C01819=1228.848,396.986,-78.994,-175.700,7.745,148.240
C01820=1228.852,396.739,-78.959,-175.700,7.743,148.239
C01821=1228.857,396.491,-78.926,-175.701,7.740,148.239
C01822=1228.860,396.243,-78.891,-175.702,7.738,148.239
C01823=1228.864,395.996,-78.857,-175.703,7.735,148.238
C01824=1228.869,395.748,-78.824,-175.703,7.733,148.238
C01825=1228.873,395.501,-78.790,-175.704,7.731,148.237
C01826=1228.876,395.253,-78.755,-175.705,7.728,148.237
C01827=1228.881,395.005,-78.722,-175.706,7.726,148.237
C01828=1228.885,394.758,-78.688,-175.707,7.723,148.236
C01829=1228.890,394.510,-78.654,-175.707,7.721,148.236
C01830=1228.893,394.262,-78.620,-175.708,7.718,148.235
C01831=1228.897,394.015,-78.586,-175.709,7.716,148.235
C01832=1228.902,393.767,-78.552,-175.710,7.713,148.234
C01833=1228.906,393.486,-78.513,-175.711,7.711,148.234
C01834=1228.911,393.204,-78.476,-175.712,7.707,148.233
C01835=1228.915,392.923,-78.437,-175.713,7.706,148.233
C01836=1228.920,392.641,-78.398,-175.714,7.703,148.233
C01837=1228.924,392.394,-78.364,-175.714,7.700,148.232
C01838=1228.928,392.147,-78.330,-175.715,7.698,148.232
C01839=1228.933,391.899,-78.297,-175.716,7.695,148.231
C01840=1228.936,391.651,-78.262,-175.717,7.692,148.231
C01841=1228.940,391.403,-78.229,-175.718,7.690,148.231
C01842=1228.945,391.156,-78.195,-175.719,7.687,148.230
C01843=1228.949,390.908,-78.161,-175.720,7.685,148.230
C01844=1228.952,390.660,-78.127,-175.721,7.682,148.229
C01845=1228.957,390.412,-78.093,-175.721,7.680,148.229
C01846=1228.961,390.165,-78.060,-175.722,7.677,148.229
C01847=1228.965,389.917,-78.026,-175.723,7.675,148.228
C01848=1228.970,389.670,-77.992,-175.724,7.672,148.228
C01849=1228.973,389.421,-77.958,-175.725,7.670,148.227
C01850=1228.977,389.174,-77.925,-175.726,7.668,148.227
C01851=1228.981,388.926,-77.891,-175.727,7.665,148.227
C01852=1228.986,388.679,-77.857,-175.728,7.663,148.226
C01853=1228.990,388.431,-77.824,-175.729,7.660,148.226
C01854=1228.993,388.183,-77.790,-175.730,7.657,148.225
C01855=1228.998,387.935,-77.756,-175.730,7.655,148.225
C01856=1229.002,387.688,-77.723,-175.731,7.652,148.225
C01857=1229.006,387.441,-77.689,-175.733,7.649,148.224
C01858=1229.010,387.193,-77.656,-175.733,7.647,148.224
C01859=1229.014,386.945,-77.621,-175.734,7.644,148.223
C01860=1229.018,386.697,-77.588,-175.736,7.642,148.223
C01861=1229.022,386.449,-77.555,-175.736,7.640,148.223
C01862=1229.026,386.202,-77.521,-175.737,7.637,148.222
C01863=1229.031,385.954,-77.487,-175.738,7.635,148.222
C01864=1229.035,385.706,-77.454,-175.739,7.632,148.222
C01865=1229.038,385.459,-77.420,-175.740,7.629,148.221
C01866=1229.042,385.211,-77.386,-175.741,7.626,148.221
C01867=1229.047,384.963,-77.353,-175.742,7.624,148.220
C01868=1229.051,384.716,-77.319,-175.743,7.622,148.220
C01869=1229.055,384.468,-77.286,-175.744,7.619,148.220
C01870=1229.059,384.220,-77.252,-175.745,7.617,148.219
C01871=1229.064,383.973,-77.218,-175.746,7.614,148.219
C01872=1229.068,383.724,-77.184,-175.747,7.611,148.218
C01873=1229.072,383.477,-77.151,-175.748,7.609,148.218
C01874=1229.075,383.230,-77.117,-175.749,7.606,148.218
C01875=1229.080,382.982,-77.084,-175.750,7.603,148.217
C01876=1229.084,382.734,-77.051,-175.752,7.601,148.217
C01877=1229.089,382.486,-77.017,-175.752,7.599,148.217
C01878=1229.092,382.239,-76.983,-175.753,7.596,148.216
C01879=1229.096,381.991,-76.950,-175.754,7.593,148.216
C01880=1229.100,381.743,-76.917,-175.756,7.590,148.215
C01881=1229.104,381.495,-76.884,-175.756,7.588,148.215
C01882=1229.108,381.248,-76.850,-175.757,7.585,148.215
C01883=1229.113,381.000,-76.816,-175.759,7.583,148.214
C01884=1229.117,380.752,-76.783,-175.760,7.580,148.214
C01885=1229.121,380.504,-76.750,-175.760,7.578,148.214
C01886=1229.125,380.257,-76.717,-175.762,7.575,148.213
C01887=1229.129,380.010,-76.683,-175.763,7.572,148.213
C01888=1229.133,379.762,-76.650,-175.764,7.570,148.213
C01889=1229.137,379.513,-76.616,-175.765,7.568,148.212
C01890=1229.142,379.265,-76.582,-175.766,7.565,148.212
C01891=1229.146,379.018,-76.549,-175.767,7.562,148.211
C01892=1229.150,378.770,-76.516,-175.768,7.559,148.211
C01893=1229.154,378.522,-76.483,-175.770,7.556,148.211
C01894=1229.158,378.275,-76.449,-175.770,7.554,148.210
C01895=1229.162,378.027,-76.416,-175.771,7.551,148.210
C01896=1229.166,377.780,-76.383,-175.773,7.549,148.210
C01897=1229.170,377.532,-76.349,-175.774,7.546,148.209
C01898=1229.175,377.284,-76.316,-175.775,7.543,148.209
C01899=1229.179,377.036,-76.283,-175.777,7.540,148.208
C01900=1229.183,376.789,-76.250,-175.777,7.539,148.208
C01901=1229.187,376.541,-76.217,-175.778,7.536,148.208
C01902=1229.191,376.293,-76.184,-175.780,7.533,148.208
C01903=1229.195,376.045,-76.150,-175.781,7.530,148.207
C01904=1229.200,375.797,-76.116,-175.782,7.528,148.207
C01905=1229.204,375.549,-76.083,-175.783,7.525,148.206
C01906=1229.208,375.301,-76.050,-175.785,7.522,148.206
C01907=1229.212,375.054,-76.017,-175.786,7.519,148.206
C01908=1229.216,374.806,-75.984,-175.787,7.517,148.205
C01909=1229.220,374.558,-75.951,-175.788,7.515,148.205
C01910=1229.224,374.310,-75.917,-175.789,7.512,148.205
C01911=1229.229,374.063,-75.884,-175.791,7.509,148.204
C01912=1229.233,373.815,-75.851,-175.792,7.506,148.204
C01913=1229.237,373.567,-75.818,-175.793,7.504,148.204
C01914=1229.241,373.320,-75.785,-175.794,7.501,148.203
C01915=1229.245,373.072,-75.752,-175.796,7.498,148.203
C01916=1229.248,372.824,-75.719,-175.797,7.495,148.203
C01917=1229.253,372.577,-75.686,-175.798,7.493,148.202
C01918=1229.257,372.329,-75.653,-175.800,7.490,148.202
C01919=1229.261,372.081,-75.620,-175.801,7.488,148.202
C01920=1229.265,371.833,-75.586,-175.802,7.485,148.201
C01921=1229.269,371.586,-75.553,-175.803,7.483,148.201
C01922=1229.274,371.337,-75.521,-175.804,7.480,148.201
C01923=1229.278,371.090,-75.488,-175.806,7.477,148.200
C01924=1229.282,370.842,-75.455,-175.807,7.474,148.200
C01925=1229.286,370.594,-75.421,-175.808,7.472,148.200
C01926=1229.290,370.346,-75.388,-175.810,7.469,148.199
C01927=1229.294,370.099,-75.355,-175.811,7.466,148.199
C01928=1229.298,369.851,-75.322,-175.812,7.463,148.199
C01929=1229.303,369.603,-75.290,-175.814,7.461,148.198
C01930=1229.306,369.355,-75.257,-175.815,7.458,148.198
C01931=1229.310,369.108,-75.224,-175.816,7.455,148.198
C01932=1229.315,368.860,-75.191,-175.818,7.453,148.198
C01933=1229.319,368.612,-75.157,-175.819,7.450,148.197
C01934=1229.324,368.364,-75.125,-175.821,7.447,148.197
C01935=1229.328,368.117,-75.092,-175.822,7.445,148.197
C01936=1229.332,367.869,-75.059,-175.823,7.442,148.196
C01937=1229.336,367.589,-75.023,-175.825,7.439,148.196
C01938=1229.341,367.309,-74.985,-175.826,7.436,148.196
C01939=1229.345,367.030,-74.948,-175.828,7.433,148.195
C01940=1229.351,366.750,-74.911,-175.830,7.429,148.195
C01941=1229.354,366.503,-74.879,-175.831,7.427,148.195
C01942=1229.358,366.255,-74.846,-175.833,7.424,148.194
C01943=1229.363,366.008,-74.812,-175.834,7.421,148.194
C01944=1229.367,365.759,-74.780,-175.835,7.419,148.194
C01945=1229.371,365.511,-74.747,-175.837,7.416,148.194
C01946=1229.375,365.264,-74.714,-175.838,7.413,148.193
C01947=1229.379,365.016,-74.682,-175.840,7.411,148.193
C01948=1229.383,364.768,-74.649,-175.841,7.408,148.193
C01949=1229.388,364.520,-74.616,-175.843,7.405,148.192
C01950=1229.392,364.272,-74.583,-175.844,7.403,148.192
C01951=1229.396,364.025,-74.551,-175.845,7.400,148.192
C01952=1229.400,363.777,-74.519,-175.847,7.398,148.192
C01953=1229.404,363.529,-74.485,-175.848,7.395,148.191
C01954=1229.409,363.281,-74.453,-175.850,7.392,148.191
C01955=1229.412,363.033,-74.420,-175.851,7.388,148.191
C01956=1229.416,362.786,-74.387,-175.853,7.386,148.190
C01957=1229.421,362.537,-74.355,-175.855,7.383,148.190
C01958=1229.424,362.290,-74.322,-175.856,7.381,148.190
C01959=1229.429,362.042,-74.290,-175.857,7.378,148.190
C01960=1229.433,361.794,-74.257,-175.859,7.375,148.189
C01961=1229.438,361.546,-74.225,-175.860,7.373,148.189
C01962=1229.441,361.299,-74.192,-175.862,7.370,148.189
C01963=1229.446,361.050,-74.160,-175.863,7.367,148.188
C01964=1229.450,360.803,-74.126,-175.865,7.365,148.188
C01965=1229.453,360.555,-74.095,-175.867,7.361,148.188
C01966=1229.458,360.308,-74.062,-175.868,7.359,148.188
C01967=1229.463,360.059,-74.029,-175.870,7.356,148.187
C01968=1229.466,359.812,-73.997,-175.871,7.354,148.187
C01969=1229.470,359.563,-73.964,-175.873,7.351,148.187
C01970=1229.475,359.315,-73.932,-175.874,7.348,148.187
C01971=1229.478,359.068,-73.899,-175.876,7.346,148.186
C01972=1229.483,358.820,-73.867,-175.877,7.343,148.186
C01973=1229.487,358.573,-73.835,-175.879,7.340,148.186
C01974=1229.491,358.324,-73.802,-175.881,7.337,148.186
C01975=1229.496,358.076,-73.770,-175.882,7.334,148.185
C01976=1229.499,357.828,-73.737,-175.884,7.332,148.185
C01977=1229.504,357.581,-73.705,-175.886,7.329,148.185
C01978=1229.507,357.333,-73.673,-175.887,7.327,148.185
C01979=1229.512,357.085,-73.640,-175.888,7.324,148.185
C01980=1229.516,356.837,-73.608,-175.890,7.321,148.184
C01981=1229.520,356.590,-73.576,-175.892,7.318,148.184
C01982=1229.525,356.342,-73.543,-175.894,7.316,148.184
C01983=1229.529,356.094,-73.511,-175.895,7.313,148.184
C01984=1229.533,355.845,-73.479,-175.896,7.310,148.183
C01985=1229.536,355.598,-73.446,-175.898,7.308,148.183
C01986=1229.541,355.350,-73.414,-175.900,7.304,148.183
C01987=1229.546,355.102,-73.382,-175.902,7.302,148.183
C01988=1229.550,354.854,-73.350,-175.904,7.299,148.183
C01989=1229.554,354.606,-73.317,-175.905,7.297,148.182
C01990=1229.558,354.359,-73.285,-175.907,7.294,148.182
C01991=1229.562,354.110,-73.253,-175.908,7.291,148.182
C01992=1229.566,353.862,-73.221,-175.910,7.288,148.182
C01993=1229.570,353.615,-73.188,-175.912,7.285,148.181
C01994=1229.575,353.367,-73.156,-175.913,7.283,148.181
C01995=1229.579,353.119,-73.124,-175.915,7.280,148.181
C01996=1229.583,352.871,-73.092,-175.917,7.278,148.181
C01997=1229.588,352.623,-73.060,-175.919,7.275,148.181
C01998=1229.592,352.375,-73.028,-175.920,7.272,148.180
C01999=1229.596,352.127,-72.995,-175.922,7.269,148.180
C02000=1229.599,351.879,-72.963,-175.924,7.267,148.180
C02001=1229.604,351.632,-72.932,-175.925,7.264,148.180
C02002=1229.608,351.384,-72.899,-175.927,7.262,148.180
C02003=1229.612,351.136,-72.867,-175.929,7.258,148.179
C02004=1229.617,350.888,-72.835,-175.931,7.256,148.179
C02005=1229.621,350.640,-72.803,-175.932,7.253,148.179
C02006=1229.625,350.392,-72.771,-175.934,7.251,148.179
C02007=1229.629,350.144,-72.739,-175.936,7.248,148.179
C02008=1229.633,349.896,-72.708,-175.938,7.245,148.178
C02009=1229.637,349.648,-72.675,-175.939,7.242,148.178
C02010=1229.642,349.401,-72.644,-175.941,7.240,148.178
C02011=1229.646,349.152,-72.611,-175.943,7.237,148.178
C02012=1229.650,348.904,-72.579,-175.945,7.234,148.178
C02013=1229.654,348.657,-72.548,-175.946,7.232,148.177
C02014=1229.659,348.409,-72.516,-175.948,7.229,148.177
C02015=1229.662,348.160,-72.484,-175.950,7.226,148.177
C02016=1229.667,347.913,-72.452,-175.951,7.224,148.177
C02017=1229.671,347.665,-72.420,-175.953,7.221,148.177
C02018=1229.675,347.417,-72.388,-175.955,7.218,148.177
C02019=1229.679,347.169,-72.356,-175.957,7.216,148.176
C02020=1229.684,346.921,-72.324,-175.958,7.213,148.176
C02021=1229.688,346.674,-72.293,-175.960,7.210,148.176
C02022=1229.692,346.426,-72.261,-175.963,7.207,148.176
C02023=1229.696,346.177,-72.228,-175.964,7.205,148.176
C02024=1229.700,345.930,-72.197,-175.966,7.202,148.176
C02025=1229.704,345.681,-72.166,-175.968,7.200,148.175
C02026=1229.709,345.433,-72.133,-175.970,7.196,148.175
C02027=1229.713,345.186,-72.102,-175.971,7.194,148.175
C02028=1229.717,344.938,-72.070,-175.973,7.191,148.175
C02029=1229.722,344.690,-72.038,-175.975,7.189,148.175
C02030=1229.726,344.442,-72.006,-175.977,7.186,148.175
C02031=1229.730,344.193,-71.975,-175.979,7.183,148.174
C02032=1229.734,343.946,-71.943,-175.980,7.181,148.174
C02033=1229.738,343.698,-71.911,-175.982,7.178,148.174
C02034=1229.743,343.450,-71.879,-175.984,7.175,148.174
C02035=1229.746,343.202,-71.848,-175.986,7.173,148.174
C02036=1229.751,342.954,-71.817,-175.988,7.170,148.174
C02037=1229.755,342.706,-71.785,-175.990,7.168,148.174
C02038=1229.760,342.459,-71.753,-175.992,7.164,148.173
C02039=1229.763,342.211,-71.721,-175.994,7.162,148.173
C02040=1229.767,341.962,-71.690,-175.995,7.159,148.173
C02041=1229.772,341.685,-71.655,-175.998,7.156,148.173
C02042=1229.777,341.408,-71.619,-175.999,7.153,148.173
C02043=1229.782,341.129,-71.584,-176.002,7.150,148.173
C02044=1229.787,340.852,-71.548,-176.004,7.147,148.172
C02045=1229.791,340.604,-71.517,-176.006,7.144,148.172
C02046=1229.795,340.356,-71.486,-176.007,7.142,148.172
C02047=1229.799,340.108,-71.454,-176.009,7.140,148.172
C02048=1229.804,339.860,-71.423,-176.012,7.136,148.172
C02049=1229.807,339.612,-71.391,-176.013,7.134,148.172
C02050=1229.812,339.365,-71.360,-176.015,7.132,148.172
C02051=1229.816,339.116,-71.328,-176.017,7.129,148.172
C02052=1229.821,338.869,-71.297,-176.019,7.126,148.171
C02053=1229.825,338.620,-71.265,-176.021,7.123,148.171
C02054=1229.829,338.373,-71.234,-176.023,7.121,148.171
C02055=1229.833,338.124,-71.203,-176.024,7.118,148.171
C02056=1229.837,337.877,-71.171,-176.027,7.115,148.171
C02057=1229.841,337.628,-71.140,-176.029,7.113,148.171
C02058=1229.846,337.381,-71.109,-176.030,7.110,148.171
C02059=1229.850,337.132,-71.078,-176.033,7.107,148.171
C02060=1229.854,336.885,-71.046,-176.035,7.105,148.170
C02061=1229.858,336.636,-71.015,-176.036,7.102,148.170
C02062=1229.862,336.389,-70.984,-176.038,7.100,148.170
C02063=1229.866,336.140,-70.952,-176.041,7.097,148.170
C02064=1229.871,335.893,-70.921,-176.043,7.094,148.170
C02065=1229.875,335.644,-70.890,-176.044,7.092,148.170
C02066=1229.879,335.397,-70.858,-176.046,7.089,148.170
C02067=1229.883,335.148,-70.827,-176.048,7.086,148.170
C02068=1229.887,334.901,-70.796,-176.050,7.084,148.170
C02069=1229.892,334.653,-70.765,-176.052,7.081,148.170
C02070=1229.896,334.404,-70.734,-176.054,7.078,148.169
C02071=1229.900,334.157,-70.702,-176.056,7.076,148.169
C02072=1229.904,333.908,-70.671,-176.058,7.073,148.169
C02073=1229.909,333.660,-70.640,-176.060,7.071,148.169
C02074=1229.912,333.412,-70.609,-176.062,7.068,148.169
C02075=1229.917,333.164,-70.578,-176.064,7.065,148.169
C02076=1229.922,332.916,-70.547,-176.066,7.063,148.169
C02077=1229.925,332.668,-70.515,-176.068,7.060,148.169
C02078=1229.930,332.420,-70.484,-176.070,7.057,148.169
C02079=1229.934,332.171,-70.453,-176.072,7.055,148.169
C02080=1229.938,331.924,-70.422,-176.074,7.053,148.169
C02081=1229.943,331.676,-70.391,-176.076,7.049,148.168
C02082=1229.947,331.427,-70.360,-176.078,7.047,148.168
C02083=1229.952,331.179,-70.329,-176.080,7.044,148.168
C02084=1229.955,330.932,-70.298,-176.082,7.042,148.168
C02085=1229.959,330.684,-70.267,-176.084,7.039,148.168
C02086=1229.964,330.436,-70.236,-176.086,7.037,148.168
C02087=1229.968,330.188,-70.206,-176.088,7.034,148.168
C02088=1229.972,329.939,-70.175,-176.091,7.031,148.168
C02089=1229.977,329.692,-70.143,-176.093,7.029,148.168
C02090=1229.981,329.443,-70.112,-176.094,7.026,148.168
C02091=1229.985,329.196,-70.082,-176.096,7.024,148.168
C02092=1229.989,328.948,-70.051,-176.099,7.021,148.168
C02093=1229.993,328.699,-70.020,-176.101,7.018,148.168
C02094=1229.998,328.451,-69.989,-176.103,7.016,148.168
C02095=1230.002,328.203,-69.958,-176.105,7.013,148.167
C02096=1230.005,327.955,-69.927,-176.107,7.011,148.167
C02097=1230.010,327.707,-69.896,-176.109,7.008,148.167
C02098=1230.015,327.459,-69.866,-176.111,7.006,148.167
C02099=1230.019,327.211,-69.835,-176.113,7.003,148.167
C02100=1230.023,326.963,-69.804,-176.115,7.000,148.167
C02101=1230.027,326.715,-69.773,-176.117,6.998,148.167
C02102=1230.032,326.467,-69.743,-176.119,6.995,148.167
C02103=1230.036,326.219,-69.712,-176.121,6.992,148.167
C02104=1230.040,325.971,-69.681,-176.124,6.990,148.167
C02105=1230.044,325.723,-69.651,-176.125,6.988,148.167
C02106=1230.048,325.474,-69.620,-176.128,6.985,148.167
C02107=1230.053,325.226,-69.589,-176.130,6.982,148.167
C02108=1230.057,324.979,-69.559,-176.132,6.980,148.167
C02109=1230.061,324.731,-69.528,-176.134,6.977,148.167
C02110=1230.065,324.482,-69.497,-176.136,6.975,148.167
C02111=1230.070,324.234,-69.466,-176.138,6.972,148.167
C02112=1230.074,323.986,-69.436,-176.141,6.969,148.167
C02113=1230.079,323.738,-69.405,-176.143,6.967,148.167
C02114=1230.083,323.490,-69.374,-176.144,6.964,148.166
C02115=1230.087,323.242,-69.344,-176.146,6.962,148.167
C02116=1230.091,322.994,-69.314,-176.149,6.959,148.166
C02117=1230.095,322.746,-69.283,-176.151,6.957,148.167
C02118=1230.099,322.497,-69.252,-176.153,6.954,148.166
C02119=1230.104,322.249,-69.222,-176.155,6.951,148.166
C02120=1230.108,322.002,-69.191,-176.157,6.949,148.166
C02121=1230.112,321.754,-69.161,-176.159,6.946,148.166
C02122=1230.117,321.505,-69.131,-176.161,6.944,148.166
C02123=1230.120,321.257,-69.100,-176.164,6.941,148.166
C02124=1230.125,321.009,-69.069,-176.166,6.939,148.166
C02125=1230.129,320.761,-69.039,-176.168,6.936,148.166
C02126=1230.134,320.513,-69.008,-176.170,6.933,148.166
C02127=1230.139,320.265,-68.978,-176.172,6.931,148.166
C02128=1230.142,320.016,-68.948,-176.174,6.929,148.166
C02129=1230.146,319.768,-68.917,-176.177,6.927,148.166
C02130=1230.150,319.521,-68.887,-176.179,6.923,148.166
C02131=1230.155,319.272,-68.857,-176.181,6.921,148.166
C02132=1230.159,319.024,-68.827,-176.183,6.919,148.166
C02133=1230.163,318.776,-68.796,-176.186,6.916,148.166
C02134=1230.167,318.528,-68.766,-176.188,6.913,148.166
C02135=1230.172,318.280,-68.735,-176.189,6.911,148.166
C02136=1230.176,318.032,-68.705,-176.191,6.909,148.166
C02137=1230.181,317.783,-68.675,-176.194,6.906,148.166
C02138=1230.185,317.536,-68.645,-176.196,6.903,148.166
C02139=1230.189,317.288,-68.614,-176.198,6.901,148.166
C02140=1230.193,317.039,-68.584,-176.201,6.898,148.166
C02141=1230.197,316.791,-68.554,-176.202,6.896,148.166
C02142=1230.202,316.543,-68.524,-176.205,6.893,148.166
C02143=1230.206,316.295,-68.493,-176.207,6.891,148.166
C02144=1230.210,316.047,-68.463,-176.209,6.888,148.166
C02145=1230.215,315.771,-68.430,-176.211,6.886,148.166
C02146=1230.220,315.496,-68.396,-176.214,6.883,148.166
C02147=1230.225,315.219,-68.363,-176.217,6.880,148.166
C02148=1230.229,314.944,-68.329,-176.219,6.878,148.166
C02149=1230.234,314.695,-68.299,-176.221,6.874,148.166
C02150=1230.238,314.448,-68.269,-176.224,6.872,148.166
C02151=1230.242,314.199,-68.239,-176.226,6.870,148.166
C02152=1230.247,313.951,-68.209,-176.227,6.867,148.166
C02153=1230.251,313.703,-68.179,-176.230,6.864,148.166
C02154=1230.256,313.455,-68.149,-176.232,6.862,148.166
C02155=1230.259,313.207,-68.119,-176.234,6.860,148.166
C02156=1230.264,312.959,-68.089,-176.237,6.857,148.166
C02157=1230.268,312.711,-68.059,-176.239,6.855,148.166
C02158=1230.272,312.462,-68.029,-176.241,6.852,148.166
C02159=1230.276,312.214,-67.999,-176.243,6.850,148.166
C02160=1230.281,311.966,-67.969,-176.246,6.847,148.166
C02161=1230.285,311.717,-67.939,-176.248,6.845,148.166
C02162=1230.289,311.470,-67.909,-176.250,6.843,148.166
C02163=1230.294,311.221,-67.879,-176.253,6.840,148.166
C02164=1230.298,310.973,-67.850,-176.255,6.837,148.166
C02165=1230.302,310.725,-67.819,-176.257,6.835,148.167
C02166=1230.307,310.477,-67.789,-176.259,6.833,148.167
C02167=1230.311,310.228,-67.760,-176.262,6.830,148.167
C02168=1230.315,309.981,-67.730,-176.264,6.828,148.167
C02169=1230.320,309.732,-67.700,-176.266,6.825,148.167
C02170=1230.324,309.484,-67.670,-176.268,6.822,148.167
C02171=1230.328,309.236,-67.641,-176.271,6.820,148.167
C02172=1230.332,308.988,-67.611,-176.273,6.818,148.167
C02173=1230.337,308.739,-67.581,-176.275,6.816,148.167
C02174=1230.341,308.491,-67.551,-176.277,6.813,148.167
C02175=1230.345,308.243,-67.522,-176.279,6.810,148.167
C02176=1230.349,307.995,-67.491,-176.282,6.808,148.167
C02177=1230.353,307.747,-67.462,-176.284,6.806,148.167
C02178=1230.358,307.498,-67.432,-176.286,6.803,148.167
C02179=1230.362,307.250,-67.403,-176.288,6.801,148.167
C02180=1230.366,307.002,-67.373,-176.291,6.799,148.167
C02181=1230.371,306.753,-67.344,-176.293,6.796,148.167
C02182=1230.375,306.507,-67.314,-176.295,6.793,148.167
C02183=1230.380,306.258,-67.284,-176.297,6.791,148.167
C02184=1230.384,306.010,-67.254,-176.300,6.789,148.167
C02185=1230.388,305.761,-67.225,-176.302,6.786,148.167
C02186=1230.393,305.513,-67.195,-176.304,6.784,148.167
C02187=1230.397,305.265,-67.166,-176.306,6.781,148.167
C02188=1230.401,305.017,-67.137,-176.308,6.779,148.167
C02189=1230.406,304.768,-67.106,-176.311,6.776,148.167
C02190=1230.410,304.520,-67.077,-176.313,6.774,148.167
C02191=1230.414,304.271,-67.048,-176.315,6.772,148.168
C02192=1230.418,304.023,-67.018,-176.318,6.770,148.168
C02193=1230.423,303.775,-66.989,-176.321,6.767,148.168
C02194=1230.427,303.527,-66.960,-176.323,6.764,148.168
C02195=1230.431,303.279,-66.930,-176.325,6.762,148.168
C02196=1230.436,303.031,-66.901,-176.327,6.760,148.168
C02197=1230.440,302.783,-66.871,-176.330,6.757,148.168
C02198=1230.444,302.534,-66.842,-176.332,6.755,148.168
C02199=1230.448,302.286,-66.812,-176.334,6.752,148.168
C02200=1230.452,302.038,-66.783,-176.336,6.750,148.168
C02201=1230.457,301.789,-66.753,-176.339,6.747,148.168
C02202=1230.462,301.541,-66.723,-176.341,6.745,148.168
C02203=1230.466,301.293,-66.694,-176.343,6.743,148.168
C02204=1230.470,301.045,-66.665,-176.345,6.741,148.169
C02205=1230.475,300.797,-66.635,-176.348,6.738,148.169
C02206=1230.479,300.548,-66.607,-176.350,6.736,148.169
C02207=1230.483,300.300,-66.577,-176.352,6.733,148.169
C02208=1230.488,300.051,-66.548,-176.355,6.731,148.169
C02209=1230.492,299.804,-66.519,-176.357,6.728,148.169
C02210=1230.496,299.556,-66.489,-176.360,6.726,148.169
C02211=1230.500,299.308,-66.460,-176.362,6.724,148.169
C02212=1230.504,299.059,-66.432,-176.364,6.722,148.169
C02213=1230.509,298.810,-66.402,-176.367,6.719,148.169
C02214=1230.513,298.563,-66.373,-176.369,6.717,148.169
C02215=1230.518,298.315,-66.344,-176.371,6.714,148.169
C02216=1230.522,298.066,-66.314,-176.373,6.712,148.170
C02217=1230.526,297.817,-66.285,-176.376,6.709,148.170
C02218=1230.530,297.569,-66.256,-176.378,6.707,148.170
C02219=1230.535,297.321,-66.226,-176.381,6.705,148.170
C02220=1230.540,297.073,-66.198,-176.383,6.703,148.170
C02221=1230.544,296.824,-66.169,-176.385,6.700,148.170
C02222=1230.548,296.576,-66.139,-176.387,6.698,148.170
C02223=1230.551,296.328,-66.110,-176.390,6.696,148.170
C02224=1230.557,296.080,-66.082,-176.392,6.693,148.170
C02225=1230.561,295.832,-66.053,-176.394,6.691,148.170
C02226=1230.565,295.583,-66.024,-176.397,6.688,148.170
C02227=1230.569,295.335,-65.994,-176.399,6.686,148.171
C02228=1230.574,295.087,-65.965,-176.402,6.684,148.171
C02229=1230.579,294.838,-65.936,-176.404,6.682,148.171
C02230=1230.582,294.590,-65.908,-176.406,6.679,148.171
C02231=1230.586,294.342,-65.878,-176.409,6.677,148.171
C02232=1230.591,294.094,-65.850,-176.411,6.675,148.171
C02233=1230.596,293.846,-65.820,-176.413,6.672,148.171
C02234=1230.600,293.597,-65.792,-176.415,6.670,148.171
C02235=1230.604,293.349,-65.763,-176.418,6.667,148.171
C02236=1230.609,293.100,-65.734,-176.420,6.665,148.172
C02237=1230.613,292.852,-65.705,-176.423,6.663,148.172
C02238=1230.617,292.603,-65.676,-176.425,6.661,148.172
C02239=1230.621,292.356,-65.648,-176.428,6.658,148.172
C02240=1230.626,292.107,-65.619,-176.430,6.656,148.172
C02241=1230.630,291.859,-65.590,-176.432,6.654,148.172
C02242=1230.635,291.611,-65.561,-176.435,6.652,148.172
C02243=1230.639,291.363,-65.532,-176.437,6.649,148.172
C02244=1230.643,291.114,-65.504,-176.439,6.646,148.172
C02245=1230.647,290.866,-65.474,-176.442,6.644,148.173
C02246=1230.652,290.617,-65.446,-176.444,6.642,148.173
C02247=1230.656,290.369,-65.418,-176.446,6.640,148.173
C02248=1230.661,290.121,-65.388,-176.448,6.638,148.173
C02249=1230.666,289.847,-65.357,-176.451,6.635,148.173
C02250=1230.670,289.573,-65.325,-176.454,6.633,148.173
C02251=1230.675,289.298,-65.294,-176.457,6.630,148.173
C02252=1230.680,289.024,-65.261,-176.459,6.627,148.173
C02253=1230.684,288.777,-65.233,-176.462,6.625,148.174
C02254=1230.689,288.528,-65.205,-176.464,6.623,148.174
C02255=1230.692,288.280,-65.176,-176.466,6.621,148.174
C02256=1230.697,288.032,-65.147,-176.469,6.619,148.174
C02257=1230.702,287.783,-65.119,-176.471,6.616,148.174
C02258=1230.706,287.535,-65.091,-176.473,6.614,148.174
C02259=1230.710,287.287,-65.061,-176.476,6.612,148.174
C02260=1230.715,287.038,-65.033,-176.478,6.609,148.175
C02261=1230.719,286.790,-65.005,-176.481,6.608,148.175
C02262=1230.723,286.541,-64.976,-176.483,6.605,148.175
C02263=1230.727,286.294,-64.948,-176.486,6.602,148.175
C02264=1230.732,286.045,-64.919,-176.488,6.600,148.175
C02265=1230.736,285.796,-64.891,-176.490,6.598,148.175
C02266=1230.741,285.548,-64.862,-176.492,6.596,148.175
C02267=1230.745,285.299,-64.834,-176.495,6.594,148.176
C02268=1230.749,285.052,-64.805,-176.498,6.591,148.176
C02269=1230.754,284.803,-64.777,-176.500,6.589,148.176
C02270=1230.758,284.555,-64.749,-176.502,6.587,148.176
C02271=1230.763,284.306,-64.720,-176.504,6.585,148.176
C02272=1230.767,284.058,-64.692,-176.507,6.583,148.176
C02273=1230.771,283.809,-64.663,-176.509,6.580,148.176
C02274=1230.775,283.561,-64.635,-176.512,6.578,148.177
C02275=1230.780,283.313,-64.607,-176.514,6.576,148.177
C02276=1230.784,283.064,-64.579,-176.517,6.574,148.177
C02277=1230.789,282.817,-64.550,-176.519,6.571,148.177
C02278=1230.793,282.568,-64.522,-176.521,6.569,148.177
C02279=1230.798,282.320,-64.493,-176.524,6.567,148.177
C02280=1230.801,282.071,-64.465,-176.526,6.564,148.177
C02281=1230.807,281.823,-64.437,-176.529,6.562,148.178
C02282=1230.810,281.574,-64.409,-176.531,6.560,148.178
C02283=1230.815,281.327,-64.381,-176.534,6.558,148.178
C02284=1230.819,281.078,-64.352,-176.536,6.556,148.178
C02285=1230.823,280.830,-64.324,-176.538,6.554,148.178
C02286=1230.828,280.581,-64.296,-176.541,6.551,148.178
C02287=1230.832,280.333,-64.268,-176.543,6.549,148.178
C02288=1230.836,280.084,-64.240,-176.546,6.547,148.179
C02289=1230.841,279.836,-64.212,-176.548,6.545,148.179
C02290=1230.845,279.587,-64.184,-176.550,6.543,148.179
C02291=1230.850,279.339,-64.155,-176.553,6.541,148.179
C02292=1230.854,279.090,-64.127,-176.556,6.538,148.179
C02293=1230.858,278.842,-64.100,-176.558,6.536,148.179
C02294=1230.863,278.594,-64.071,-176.560,6.534,148.180
C02295=1230.867,278.346,-64.043,-176.563,6.532,148.180
C02296=1230.872,278.098,-64.015,-176.565,6.530,148.180
C02297=1230.876,277.848,-63.987,-176.567,6.527,148.180
C02298=1230.881,277.600,-63.959,-176.570,6.526,148.181
C02299=1230.884,277.352,-63.931,-176.573,6.522,148.181
C02300=1230.890,277.104,-63.903,-176.575,6.521,148.181
C02301=1230.893,276.855,-63.875,-176.577,6.518,148.181
C02302=1230.898,276.607,-63.847,-176.580,6.516,148.181
C02303=1230.902,276.359,-63.820,-176.582,6.514,148.181
C02304=1230.907,276.110,-63.791,-176.585,6.512,148.182
C02305=1230.911,275.862,-63.763,-176.587,6.510,148.182
C02306=1230.915,275.613,-63.735,-176.589,6.508,148.182
C02307=1230.920,275.365,-63.708,-176.592,6.505,148.182
C02308=1230.925,275.117,-63.680,-176.595,6.503,148.182
C02309=1230.928,274.868,-63.652,-176.597,6.501,148.182
C02310=1230.933,274.620,-63.625,-176.599,6.499,148.183
C02311=1230.938,274.371,-63.596,-176.601,6.497,148.183
C02312=1230.942,274.123,-63.568,-176.604,6.495,148.183
C02313=1230.947,273.874,-63.541,-176.606,6.493,148.183
C02314=1230.950,273.626,-63.513,-176.609,6.491,148.183
C02315=1230.955,273.378,-63.485,-176.611,6.488,148.183
C02316=1230.960,273.129,-63.458,-176.614,6.486,148.184
C02317=1230.964,272.881,-63.429,-176.617,6.484,148.184
C02318=1230.968,272.633,-63.402,-176.619,6.482,148.184
C02319=1230.972,272.383,-63.374,-176.621,6.480,148.184
C02320=1230.977,272.136,-63.346,-176.623,6.478,148.184
C02321=1230.981,271.887,-63.319,-176.626,6.476,148.185
C02322=1230.986,271.638,-63.291,-176.628,6.474,148.185
C02323=1230.990,271.390,-63.264,-176.631,6.472,148.185
C02324=1230.995,271.142,-63.236,-176.634,6.469,148.185
C02325=1230.999,270.893,-63.209,-176.636,6.467,148.185
C02326=1231.003,270.645,-63.181,-176.639,6.465,148.186
C02327=1231.008,270.396,-63.153,-176.641,6.463,148.186
C02328=1231.012,270.148,-63.126,-176.643,6.461,148.186
C02329=1231.016,269.899,-63.098,-176.645,6.459,148.186
C02330=1231.021,269.651,-63.070,-176.648,6.457,148.186
C02331=1231.026,269.402,-63.043,-176.651,6.455,148.187
C02332=1231.030,269.154,-63.015,-176.653,6.453,148.187
C02333=1231.034,268.905,-62.988,-176.655,6.451,148.187
C02334=1231.039,268.658,-62.960,-176.658,6.448,148.187
C02335=1231.043,268.409,-62.933,-176.661,6.446,148.187
C02336=1231.047,268.160,-62.905,-176.663,6.444,148.188
C02337=1231.052,267.912,-62.878,-176.665,6.442,148.188
C02338=1231.056,267.663,-62.851,-176.668,6.440,148.188
C02339=1231.061,267.416,-62.823,-176.670,6.438,148.188
C02340=1231.065,267.166,-62.795,-176.673,6.436,148.188
C02341=1231.069,266.918,-62.768,-176.675,6.434,148.189
C02342=1231.074,266.670,-62.740,-176.677,6.432,148.189
C02343=1231.078,266.422,-62.713,-176.680,6.430,148.189
C02344=1231.083,266.172,-62.686,-176.682,6.427,148.189
C02345=1231.087,265.924,-62.658,-176.685,6.426,148.189
C02346=1231.092,265.676,-62.631,-176.687,6.424,148.190
C02347=1231.096,265.427,-62.604,-176.690,6.421,148.190
C02348=1231.101,265.179,-62.577,-176.692,6.419,148.190
C02349=1231.105,264.930,-62.549,-176.695,6.417,148.190
C02350=1231.109,264.682,-62.522,-176.697,6.415,148.190
C02351=1231.114,264.433,-62.495,-176.700,6.413,148.191
C02352=1231.119,264.185,-62.468,-176.702,6.411,148.191
C02353=1231.123,263.913,-62.438,-176.704,6.409,148.191
C02354=1231.128,263.640,-62.408,-176.708,6.406,148.191
C02355=1231.132,263.367,-62.378,-176.710,6.404,148.192
C02356=1231.137,263.095,-62.348,-176.713,6.402,148.192
C02357=1231.141,262.846,-62.321,-176.715,6.400,148.192
C02358=1231.146,262.598,-62.294,-176.718,6.398,148.192
C02359=1231.151,262.349,-62.267,-176.720,6.396,148.193
C02360=1231.155,262.101,-62.240,-176.723,6.393,148.193
C02361=1231.160,261.852,-62.213,-176.725,6.391,148.193
C02362=1231.163,261.603,-62.186,-176.728,6.389,148.193
C02363=1231.168,261.355,-62.158,-176.730,6.387,148.193
C02364=1231.172,261.107,-62.131,-176.733,6.385,148.194
C02365=1231.177,260.858,-62.104,-176.735,6.383,148.194
C02366=1231.182,260.610,-62.077,-176.738,6.381,148.194
C02367=1231.186,260.361,-62.050,-176.740,6.379,148.194
C02368=1231.190,260.113,-62.023,-176.743,6.377,148.195
C02369=1231.194,259.864,-61.996,-176.745,6.375,148.195
C02370=1231.199,259.616,-61.969,-176.747,6.373,148.195
C02371=1231.204,259.367,-61.942,-176.750,6.371,148.195
C02372=1231.208,259.119,-61.915,-176.753,6.369,148.196
C02373=1231.212,258.870,-61.888,-176.755,6.367,148.196
C02374=1231.217,258.622,-61.861,-176.757,6.365,148.196
C02375=1231.222,258.373,-61.834,-176.760,6.363,148.196
C02376=1231.226,258.125,-61.807,-176.762,6.361,148.196
C02377=1231.230,257.877,-61.781,-176.765,6.359,148.197
C02378=1231.235,257.628,-61.753,-176.767,6.357,148.197
C02379=1231.239,257.379,-61.726,-176.770,6.355,148.197
C02380=1231.244,257.131,-61.699,-176.772,6.353,148.197
C02381=1231.248,256.882,-61.673,-176.775,6.351,148.198
C02382=1231.252,256.633,-61.646,-176.777,6.349,148.198
C02383=1231.257,256.385,-61.619,-176.779,6.347,148.198
C02384=1231.261,256.137,-61.593,-176.782,6.345,148.198
C02385=1231.266,255.888,-61.566,-176.785,6.343,148.199
C02386=1231.270,255.640,-61.539,-176.787,6.342,148.199
C02387=1231.274,255.391,-61.512,-176.789,6.339,148.199
C02388=1231.279,255.142,-61.486,-176.792,6.337,148.199
C02389=1231.284,254.894,-61.459,-176.794,6.336,148.200
C02390=1231.288,254.646,-61.432,-176.797,6.334,148.200
C02391=1231.292,254.397,-61.405,-176.799,6.332,148.200
C02392=1231.297,254.149,-61.378,-176.802,6.330,148.200
C02393=1231.301,253.900,-61.352,-176.804,6.328,148.201
C02394=1231.306,253.651,-61.325,-176.807,6.326,148.201
C02395=1231.311,253.403,-61.298,-176.809,6.324,148.201
C02396=1231.315,253.155,-61.272,-176.812,6.322,148.201
C02397=1231.319,252.905,-61.245,-176.814,6.320,148.202
C02398=1231.323,252.657,-61.219,-176.817,6.318,148.202
C02399=1231.328,252.409,-61.192,-176.819,6.316,148.202
C02400=1231.333,252.160,-61.165,-176.822,6.314,148.202
C02401=1231.337,251.912,-61.139,-176.824,6.312,148.203
C02402=1231.342,251.663,-61.112,-176.827,6.310,148.203
C02403=1231.346,251.415,-61.085,-176.829,6.308,148.203
C02404=1231.350,251.166,-61.059,-176.832,6.306,148.203
C02405=1231.354,250.918,-61.033,-176.834,6.304,148.204
C02406=1231.359,250.668,-61.006,-176.837,6.302,148.204
C02407=1231.363,250.420,-60.980,-176.839,6.300,148.204
C02408=1231.368,250.172,-60.953,-176.842,6.298,148.204
C02409=1231.372,249.923,-60.927,-176.844,6.296,148.205
C02410=1231.377,249.674,-60.900,-176.847,6.294,148.205
C02411=1231.381,249.426,-60.874,-176.849,6.292,148.205
C02412=1231.386,249.177,-60.847,-176.852,6.290,148.205
C02413=1231.390,248.929,-60.821,-176.854,6.288,148.206
C02414=1231.395,248.681,-60.795,-176.857,6.287,148.206
C02415=1231.399,248.432,-60.768,-176.859,6.285,148.206
C02416=1231.404,248.183,-60.742,-176.862,6.283,148.207
C02417=1231.408,247.935,-60.715,-176.864,6.281,148.207
C02418=1231.413,247.686,-60.689,-176.867,6.279,148.207
C02419=1231.417,247.438,-60.663,-176.869,6.277,148.207
C02420=1231.422,247.189,-60.636,-176.872,6.275,148.208
C02421=1231.426,246.940,-60.610,-176.875,6.273,148.208
C02422=1231.430,246.692,-60.584,-176.877,6.271,148.208
C02423=1231.435,246.443,-60.558,-176.879,6.269,148.208
C02424=1231.439,246.195,-60.532,-176.882,6.267,148.209
C02425=1231.444,245.946,-60.505,-176.885,6.265,148.209
C02426=1231.448,245.698,-60.479,-176.887,6.263,148.209
C02427=1231.453,245.449,-60.453,-176.890,6.261,148.210
C02428=1231.457,245.200,-60.426,-176.892,6.259,148.210
C02429=1231.461,244.952,-60.400,-176.894,6.257,148.210
C02430=1231.466,244.703,-60.375,-176.897,6.255,148.210
C02431=1231.470,244.454,-60.347,-176.900,6.254,148.211
C02432=1231.475,244.206,-60.322,-176.902,6.252,148.211
C02433=1231.479,243.957,-60.296,-176.904,6.250,148.211
C02434=1231.484,243.709,-60.269,-176.906,6.248,148.211
C02435=1231.488,243.460,-60.244,-176.909,6.246,148.212
C02436=1231.492,243.211,-60.218,-176.912,6.245,148.212
C02437=1231.497,242.963,-60.191,-176.914,6.243,148.212
C02438=1231.502,242.715,-60.165,-176.917,6.241,148.213
C02439=1231.506,242.466,-60.140,-176.920,6.239,148.213
C02440=1231.511,242.217,-60.113,-176.922,6.237,148.213
C02441=1231.515,241.969,-60.087,-176.924,6.235,148.213
C02442=1231.519,241.720,-60.061,-176.927,6.233,148.214
C02443=1231.524,241.472,-60.036,-176.930,6.231,148.214
C02444=1231.529,241.223,-60.009,-176.932,6.229,148.214
C02445=1231.533,240.974,-59.984,-176.935,6.227,148.215
C02446=1231.537,240.726,-59.957,-176.937,6.225,148.215
C02447=1231.541,240.477,-59.931,-176.939,6.223,148.215
C02448=1231.547,240.228,-59.905,-176.942,6.222,148.215
C02449=1231.551,239.980,-59.880,-176.944,6.220,148.216
C02450=1231.555,239.731,-59.854,-176.947,6.218,148.216
C02451=1231.560,239.482,-59.828,-176.949,6.217,148.216
C02452=1231.565,239.234,-59.801,-176.952,6.215,148.217
C02453=1231.569,238.985,-59.776,-176.955,6.213,148.217
C02454=1231.573,238.737,-59.750,-176.957,6.211,148.217
C02455=1231.578,238.488,-59.724,-176.959,6.209,148.217
C02456=1231.582,238.240,-59.699,-176.962,6.207,148.218
C02457=1231.587,237.968,-59.671,-176.965,6.205,148.218
C02458=1231.592,237.697,-59.642,-176.967,6.203,148.218
C02459=1231.597,237.425,-59.614,-176.970,6.201,148.219
C02460=1231.602,237.153,-59.586,-176.973,6.198,148.219
C02461=1231.607,236.905,-59.560,-176.975,6.197,148.219
C02462=1231.611,236.656,-59.534,-176.978,6.196,148.220
C02463=1231.616,236.407,-59.509,-176.980,6.194,148.220
C02464=1231.620,236.159,-59.483,-176.983,6.192,148.220
C02465=1231.625,235.910,-59.458,-176.986,6.190,148.220
C02466=1231.629,235.662,-59.432,-176.988,6.188,148.221
C02467=1231.634,235.414,-59.406,-176.991,6.186,148.221
C02468=1231.638,235.165,-59.381,-176.993,6.184,148.221
C02469=1231.642,234.916,-59.355,-176.996,6.182,148.222
C02470=1231.647,234.667,-59.329,-176.998,6.180,148.222
C02471=1231.652,234.419,-59.303,-177.001,6.178,148.222
C02472=1231.656,234.170,-59.277,-177.003,6.177,148.223
C02473=1231.660,233.921,-59.252,-177.005,6.175,148.223
C02474=1231.665,233.673,-59.226,-177.008,6.174,148.223
C02475=1231.669,233.424,-59.201,-177.011,6.172,148.223
C02476=1231.674,233.175,-59.176,-177.013,6.170,148.224
C02477=1231.679,232.927,-59.150,-177.016,6.168,148.224
C02478=1231.683,232.678,-59.124,-177.018,6.166,148.224
C02479=1231.688,232.430,-59.099,-177.021,6.164,148.225
C02480=1231.692,232.181,-59.073,-177.024,6.162,148.225
C02481=1231.696,231.932,-59.048,-177.026,6.161,148.225
C02482=1231.701,231.683,-59.023,-177.028,6.159,148.226
C02483=1231.706,231.435,-58.997,-177.031,6.157,148.226
C02484=1231.710,231.186,-58.971,-177.033,6.155,148.226
C02485=1231.715,230.938,-58.946,-177.036,6.153,148.226
C02486=1231.719,230.688,-58.921,-177.038,6.152,148.227
C02487=1231.724,230.440,-58.896,-177.041,6.150,148.227
C02488=1231.728,230.191,-58.870,-177.044,6.148,148.227
C02489=1231.732,229.943,-58.844,-177.046,6.147,148.228
C02490=1231.738,229.694,-58.819,-177.048,6.145,148.228
C02491=1231.741,229.445,-58.794,-177.051,6.143,148.228
C02492=1231.746,229.197,-58.769,-177.054,6.141,148.229
C02493=1231.750,228.948,-58.743,-177.056,6.139,148.229
C02494=1231.755,228.700,-58.718,-177.059,6.137,148.229
C02495=1231.759,228.451,-58.693,-177.061,6.135,148.230
C02496=1231.764,228.202,-58.668,-177.064,6.134,148.230
C02497=1231.769,227.953,-58.642,-177.066,6.133,148.230
C02498=1231.773,227.705,-58.617,-177.069,6.131,148.231
C02499=1231.778,227.456,-58.592,-177.071,6.129,148.231
C02500=1231.782,227.207,-58.567,-177.074,6.127,148.231
C02501=1231.786,226.959,-58.541,-177.077,6.125,148.232
C02502=1231.791,226.710,-58.516,-177.079,6.123,148.232
C02503=1231.796,226.462,-58.491,-177.082,6.121,148.232
C02504=1231.800,226.212,-58.466,-177.083,6.120,148.232
C02505=1231.805,225.964,-58.440,-177.086,6.118,148.233
C02506=1231.809,225.715,-58.416,-177.089,6.116,148.233
C02507=1231.813,225.466,-58.390,-177.091,6.114,148.233
C02508=1231.818,225.218,-58.366,-177.094,6.112,148.234
C02509=1231.823,224.969,-58.340,-177.097,6.111,148.234
C02510=1231.828,224.720,-58.315,-177.099,6.109,148.234
C02511=1231.831,224.472,-58.290,-177.101,6.108,148.235
C02512=1231.836,224.223,-58.265,-177.104,6.106,148.235
C02513=1231.841,223.974,-58.240,-177.106,6.104,148.235
C02514=1231.846,223.725,-58.215,-177.109,6.102,148.236
C02515=1231.850,223.478,-58.190,-177.112,6.100,148.236
C02516=1231.854,223.228,-58.165,-177.114,6.098,148.236
C02517=1231.859,222.980,-58.140,-177.117,6.096,148.237
C02518=1231.864,222.731,-58.115,-177.119,6.095,148.237
C02519=1231.868,222.483,-58.090,-177.122,6.094,148.237
C02520=1231.872,222.233,-58.065,-177.124,6.092,148.238
C02521=1231.877,221.985,-58.040,-177.127,6.090,148.238
C02522=1231.881,221.736,-58.015,-177.130,6.088,148.238
C02523=1231.886,221.487,-57.990,-177.132,6.086,148.239
C02524=1231.891,221.238,-57.965,-177.134,6.085,148.239
C02525=1231.895,220.990,-57.940,-177.137,6.083,148.239
C02526=1231.900,220.741,-57.916,-177.139,6.081,148.240
C02527=1231.904,220.492,-57.891,-177.142,6.079,148.240
C02528=1231.909,220.244,-57.865,-177.145,6.078,148.241
C02529=1231.913,219.995,-57.841,-177.148,6.076,148.241
C02530=1231.918,219.746,-57.816,-177.150,6.075,148.241
C02531=1231.922,219.498,-57.791,-177.153,6.073,148.242
C02532=1231.927,219.249,-57.767,-177.155,6.071,148.242
C02533=1231.932,219.000,-57.742,-177.158,6.069,148.242
C02534=1231.936,218.751,-57.717,-177.160,6.067,148.243
C02535=1231.940,218.503,-57.692,-177.163,6.066,148.243
C02536=1231.945,218.254,-57.667,-177.165,6.065,148.243
C02537=1231.949,218.005,-57.643,-177.168,6.063,148.244
C02538=1231.954,217.756,-57.618,-177.170,6.061,148.244
C02539=1231.958,217.507,-57.594,-177.173,6.059,148.244
C02540=1231.963,217.259,-57.568,-177.176,6.057,148.245
C02541=1231.967,217.011,-57.544,-177.178,6.055,148.245
C02542=1231.972,216.761,-57.519,-177.180,6.054,148.245
C02543=1231.977,216.513,-57.495,-177.183,6.052,148.246
C02544=1231.981,216.263,-57.470,-177.186,6.050,148.246
C02545=1231.986,216.015,-57.446,-177.188,6.049,148.246
C02546=1231.990,215.767,-57.421,-177.191,6.047,148.247
C02547=1231.995,215.518,-57.396,-177.193,6.045,148.247
C02548=1231.999,215.269,-57.372,-177.195,6.044,148.247
C02549=1232.004,215.020,-57.347,-177.199,6.042,148.248
C02550=1232.008,214.771,-57.323,-177.201,6.040,148.248
C02551=1232.013,214.523,-57.298,-177.204,6.039,148.249
C02552=1232.018,214.274,-57.274,-177.206,6.037,148.249
C02553=1232.022,214.025,-57.249,-177.209,6.036,148.249
C02554=1232.026,213.776,-57.225,-177.211,6.034,148.250
C02555=1232.032,213.528,-57.200,-177.214,6.032,148.250
C02556=1232.036,213.279,-57.176,-177.216,6.030,148.250
C02557=1232.041,213.030,-57.151,-177.219,6.028,148.251
C02558=1232.045,212.781,-57.127,-177.221,6.027,148.251
C02559=1232.049,212.533,-57.103,-177.224,6.025,148.251
C02560=1232.054,212.284,-57.078,-177.226,6.023,148.252
C02561=1232.059,212.013,-57.051,-177.230,6.022,148.252
C02562=1232.063,211.743,-57.025,-177.232,6.020,148.252
C02563=1232.069,211.473,-56.999,-177.235,6.018,148.253
C02564=1232.073,211.202,-56.972,-177.237,6.016,148.253
C02565=1232.078,210.953,-56.948,-177.240,6.014,148.253
C02566=1232.083,210.705,-56.923,-177.243,6.013,148.254
C02567=1232.087,210.456,-56.899,-177.245,6.012,148.254
C02568=1232.092,210.207,-56.874,-177.248,6.010,148.255
C02569=1232.096,209.958,-56.850,-177.250,6.008,148.255
C02570=1232.101,209.709,-56.827,-177.253,6.006,148.255
C02571=1232.106,209.461,-56.802,-177.256,6.004,148.256
C02572=1232.110,209.212,-56.778,-177.258,6.003,148.256
C02573=1232.114,208.963,-56.753,-177.260,6.002,148.256
C02574=1232.119,208.714,-56.729,-177.263,6.000,148.257
C02575=1232.124,208.466,-56.705,-177.266,5.998,148.257
C02576=1232.128,208.217,-56.681,-177.268,5.997,148.258
C02577=1232.133,207.968,-56.656,-177.271,5.995,148.258
C02578=1232.137,207.719,-56.632,-177.274,5.993,148.258
C02579=1232.142,207.471,-56.608,-177.276,5.992,148.259
C02580=1232.147,207.221,-56.584,-177.279,5.990,148.259
C02581=1232.152,206.973,-56.560,-177.281,5.989,148.259
C02582=1232.155,206.724,-56.536,-177.284,5.987,148.260
C02583=1232.160,206.475,-56.511,-177.286,5.985,148.260
C02584=1232.165,206.226,-56.488,-177.289,5.983,148.260
C02585=1232.170,205.978,-56.463,-177.291,5.982,148.261
C02586=1232.174,205.729,-56.439,-177.294,5.980,148.261
C02587=1232.179,205.480,-56.416,-177.297,5.979,148.262
C02588=1232.183,205.231,-56.391,-177.299,5.977,148.262
C02589=1232.188,204.982,-56.367,-177.301,5.976,148.262
C02590=1232.192,204.733,-56.344,-177.304,5.974,148.263
C02591=1232.197,204.485,-56.319,-177.307,5.972,148.263
C02592=1232.202,204.236,-56.295,-177.309,5.970,148.263
C02593=1232.207,203.987,-56.271,-177.312,5.969,148.264
C02594=1232.211,203.739,-56.247,-177.314,5.968,148.264
C02595=1232.215,203.490,-56.223,-177.317,5.966,148.265
C02596=1232.219,203.241,-56.200,-177.319,5.965,148.265
C02597=1232.224,202.992,-56.176,-177.322,5.963,148.265
C02598=1232.229,202.743,-56.152,-177.324,5.961,148.266
C02599=1232.234,202.494,-56.127,-177.327,5.959,148.266
C02600=1232.238,202.245,-56.104,-177.330,5.958,148.267
C02601=1232.243,201.997,-56.080,-177.332,5.957,148.267
C02602=1232.248,201.748,-56.057,-177.335,5.955,148.267
C02603=1232.252,201.500,-56.033,-177.337,5.953,148.268
C02604=1232.256,201.250,-56.008,-177.340,5.952,148.268
C02605=1232.261,201.001,-55.984,-177.342,5.950,148.268
C02606=1232.266,200.752,-55.961,-177.345,5.948,148.269
C02607=1232.270,200.504,-55.937,-177.347,5.947,148.269
C02608=1232.275,200.255,-55.913,-177.350,5.946,148.270
C02609=1232.279,200.006,-55.889,-177.353,5.944,148.270
C02610=1232.284,199.757,-55.866,-177.355,5.942,148.270
C02611=1232.288,199.509,-55.842,-177.357,5.941,148.271
C02612=1232.293,199.260,-55.819,-177.360,5.939,148.271
C02613=1232.298,199.011,-55.794,-177.363,5.937,148.272
C02614=1232.302,198.762,-55.771,-177.365,5.936,148.272
C02615=1232.307,198.513,-55.748,-177.368,5.935,148.272
C02616=1232.311,198.265,-55.724,-177.371,5.933,148.273
C02617=1232.316,198.016,-55.700,-177.373,5.931,148.273
C02618=1232.320,197.767,-55.676,-177.375,5.930,148.273
C02619=1232.325,197.518,-55.653,-177.378,5.928,148.274
C02620=1232.330,197.269,-55.630,-177.381,5.926,148.274
C02621=1232.334,197.020,-55.605,-177.383,5.925,148.275
C02622=1232.338,196.771,-55.582,-177.386,5.924,148.275
C02623=1232.343,196.522,-55.558,-177.388,5.922,148.275
C02624=1232.348,196.273,-55.535,-177.390,5.921,148.276
C02625=1232.352,196.025,-55.511,-177.394,5.919,148.276
C02626=1232.357,195.776,-55.488,-177.396,5.917,148.277
C02627=1232.361,195.527,-55.464,-177.398,5.916,148.277
C02628=1232.366,195.278,-55.440,-177.401,5.914,148.277
C02629=1232.371,195.029,-55.417,-177.404,5.913,148.278
C02630=1232.376,194.781,-55.394,-177.406,5.912,148.278
C02631=1232.381,194.532,-55.370,-177.409,5.910,148.279
C02632=1232.385,194.283,-55.346,-177.411,5.908,148.279
C02633=1232.390,194.034,-55.323,-177.414,5.906,148.279
C02634=1232.394,193.785,-55.300,-177.416,5.905,148.280
C02635=1232.399,193.536,-55.276,-177.419,5.903,148.280
C02636=1232.404,193.287,-55.253,-177.422,5.902,148.281
C02637=1232.408,193.038,-55.230,-177.424,5.901,148.281
C02638=1232.412,192.790,-55.206,-177.427,5.899,148.281
C02639=1232.417,192.541,-55.183,-177.429,5.897,148.282
C02640=1232.422,192.292,-55.159,-177.431,5.896,148.282
C02641=1232.426,192.043,-55.136,-177.434,5.895,148.283
C02642=1232.431,191.794,-55.113,-177.437,5.893,148.283
C02643=1232.436,191.545,-55.089,-177.439,5.892,148.283
C02644=1232.440,191.296,-55.066,-177.442,5.890,148.284
C02645=1232.445,191.047,-55.043,-177.444,5.889,148.284
C02646=1232.449,190.799,-55.019,-177.447,5.887,148.285
C02647=1232.454,190.551,-54.996,-177.450,5.886,148.285
C02648=1232.459,190.302,-54.973,-177.452,5.885,148.285
C02649=1232.463,190.052,-54.949,-177.454,5.883,148.286
C02650=1232.468,189.803,-54.926,-177.458,5.881,148.286
C02651=1232.472,189.555,-54.903,-177.460,5.880,148.287
C02652=1232.477,189.306,-54.880,-177.462,5.878,148.287
C02653=1232.481,189.057,-54.857,-177.465,5.876,148.287
C02654=1232.486,188.808,-54.833,-177.467,5.875,148.288
C02655=1232.491,188.559,-54.810,-177.470,5.874,148.288
C02656=1232.495,188.311,-54.787,-177.473,5.872,148.289
C02657=1232.500,188.062,-54.764,-177.475,5.871,148.289
C02658=1232.505,187.813,-54.741,-177.477,5.869,148.289
C02659=1232.510,187.563,-54.717,-177.481,5.868,148.290
C02660=1232.513,187.315,-54.695,-177.483,5.867,148.290
C02661=1232.518,187.065,-54.672,-177.485,5.865,148.291
C02662=1232.523,186.816,-54.649,-177.487,5.864,148.291
C02663=1232.528,186.568,-54.626,-177.491,5.862,148.292
C02664=1232.532,186.319,-54.603,-177.493,5.860,148.292
C02665=1232.538,186.049,-54.578,-177.495,5.859,148.292
C02666=1232.543,185.779,-54.553,-177.498,5.858,148.293
C02667=1232.548,185.510,-54.528,-177.501,5.856,148.293
C02668=1232.552,185.240,-54.502,-177.504,5.854,148.294
C02669=1232.558,184.991,-54.480,-177.507,5.853,148.294
C02670=1232.562,184.743,-54.457,-177.509,5.852,148.295
C02671=1232.566,184.493,-54.434,-177.512,5.850,148.295
C02672=1232.571,184.244,-54.410,-177.514,5.849,148.295
C02673=1232.575,183.996,-54.388,-177.517,5.847,148.296
C02674=1232.581,183.747,-54.365,-177.519,5.845,148.296
C02675=1232.585,183.498,-54.343,-177.522,5.844,148.297
C02676=1232.589,183.249,-54.319,-177.525,5.843,148.297
C02677=1232.594,183.000,-54.296,-177.527,5.842,148.298
C02678=1232.598,182.751,-54.273,-177.529,5.840,148.298
C02679=1232.604,182.502,-54.251,-177.532,5.838,148.298
C02680=1232.608,182.254,-54.228,-177.535,5.837,148.299
C02681=1232.612,182.005,-54.205,-177.537,5.836,148.299
C02682=1232.617,181.755,-54.182,-177.539,5.835,148.300
C02683=1232.622,181.507,-54.160,-177.542,5.833,148.300
C02684=1232.626,181.258,-54.136,-177.545,5.831,148.301
C02685=1232.631,181.009,-54.114,-177.547,5.830,148.301
C02686=1232.635,180.759,-54.091,-177.550,5.828,148.301
C02687=1232.640,180.511,-54.069,-177.552,5.827,148.302
C02688=1232.645,180.262,-54.046,-177.555,5.826,148.302
C02689=1232.650,180.013,-54.023,-177.558,5.824,148.303
C02690=1232.654,179.764,-54.000,-177.560,5.823,148.303
C02691=1232.659,179.515,-53.978,-177.563,5.822,148.304
C02692=1232.663,179.266,-53.955,-177.565,5.820,148.304
C02693=1232.668,179.017,-53.931,-177.568,5.819,148.304
C02694=1232.673,178.769,-53.910,-177.570,5.817,148.305
C02695=1232.678,178.520,-53.886,-177.573,5.816,148.305
C02696=1232.682,178.270,-53.864,-177.576,5.814,148.306
C02697=1232.687,178.022,-53.841,-177.578,5.813,148.306
C02698=1232.691,177.773,-53.819,-177.581,5.812,148.307
C02699=1232.696,177.524,-53.796,-177.583,5.811,148.307
C02700=1232.700,177.274,-53.774,-177.586,5.809,148.307
C02701=1232.705,177.026,-53.751,-177.588,5.807,148.308
C02702=1232.710,176.777,-53.728,-177.591,5.806,148.308
C02703=1232.714,176.528,-53.706,-177.593,5.805,148.309
C02704=1232.719,176.279,-53.684,-177.596,5.804,148.309
C02705=1232.723,176.030,-53.661,-177.599,5.802,148.310
C02706=1232.728,175.781,-53.638,-177.601,5.801,148.310
C02707=1232.733,175.533,-53.616,-177.603,5.799,148.310
C02708=1232.737,175.283,-53.594,-177.606,5.798,148.311
C02709=1232.742,175.034,-53.571,-177.609,5.797,148.311
C02710=1232.747,174.786,-53.549,-177.611,5.795,148.312
C02711=1232.752,174.537,-53.526,-177.613,5.794,148.312
C02712=1232.756,174.288,-53.504,-177.616,5.792,148.313
C02713=1232.761,174.039,-53.482,-177.619,5.791,148.313
C02714=1232.765,173.790,-53.458,-177.621,5.789,148.313
C02715=1232.770,173.541,-53.437,-177.624,5.789,148.314
C02716=1232.775,173.292,-53.413,-177.626,5.787,148.314
C02717=1232.779,173.042,-53.391,-177.629,5.786,148.315
C02718=1232.784,172.794,-53.370,-177.632,5.784,148.315
C02719=1232.789,172.545,-53.346,-177.634,5.783,148.316
C02720=1232.794,172.296,-53.325,-177.636,5.782,148.316
C02721=1232.798,172.047,-53.303,-177.639,5.781,148.317
C02722=1232.803,171.799,-53.280,-177.642,5.779,148.317
C02723=1232.807,171.549,-53.258,-177.644,5.777,148.317
C02724=1232.812,171.300,-53.235,-177.647,5.777,148.318
C02725=1232.817,171.051,-53.214,-177.650,5.775,148.318
C02726=1232.821,170.802,-53.190,-177.652,5.774,148.319
C02727=1232.826,170.554,-53.169,-177.655,5.772,148.319
C02728=1232.830,170.304,-53.147,-177.657,5.771,148.320
C02729=1232.836,170.055,-53.124,-177.660,5.769,148.320
C02730=1232.840,169.807,-53.102,-177.662,5.769,148.321
C02731=1232.844,169.557,-53.080,-177.665,5.767,148.321
C02732=1232.849,169.309,-53.058,-177.667,5.766,148.322
C02733=1232.854,169.059,-53.035,-177.670,5.764,148.322
C02734=1232.859,168.811,-53.013,-177.672,5.763,148.322
C02735=1232.863,168.562,-52.991,-177.675,5.761,148.323
C02736=1232.868,168.313,-52.969,-177.677,5.761,148.323
C02737=1232.873,168.063,-52.947,-177.680,5.759,148.324
C02738=1232.878,167.815,-52.925,-177.682,5.758,148.324
C02739=1232.882,167.565,-52.903,-177.685,5.756,148.325
C02740=1232.887,167.317,-52.881,-177.687,5.755,148.325
C02741=1232.891,167.068,-52.858,-177.690,5.754,148.326
C02742=1232.896,166.819,-52.837,-177.693,5.753,148.326
C02743=1232.901,166.570,-52.814,-177.695,5.751,148.327
C02744=1232.906,166.321,-52.792,-177.697,5.750,148.327
C02745=1232.910,166.072,-52.770,-177.700,5.749,148.328
C02746=1232.915,165.823,-52.749,-177.703,5.748,148.328
C02747=1232.919,165.574,-52.727,-177.706,5.746,148.328
C02748=1232.924,165.325,-52.705,-177.708,5.745,148.329
C02749=1232.929,165.075,-52.682,-177.710,5.743,148.329
C02750=1232.934,164.827,-52.661,-177.713,5.743,148.330
C02751=1232.938,164.577,-52.639,-177.716,5.741,148.330
C02752=1232.943,164.329,-52.617,-177.718,5.740,148.331
C02753=1232.947,164.079,-52.595,-177.721,5.738,148.331
C02754=1232.952,163.831,-52.573,-177.723,5.737,148.332
C02755=1232.956,163.581,-52.551,-177.726,5.735,148.332
C02756=1232.961,163.333,-52.529,-177.728,5.735,148.333
C02757=1232.965,163.083,-52.507,-177.731,5.733,148.333
C02758=1232.970,162.835,-52.486,-177.734,5.732,148.334
C02759=1232.976,162.586,-52.463,-177.736,5.730,148.334
C02760=1232.980,162.336,-52.441,-177.738,5.729,148.334
C02761=1232.985,162.088,-52.420,-177.741,5.728,148.335
C02762=1232.989,161.838,-52.398,-177.744,5.727,148.335
C02763=1232.994,161.590,-52.376,-177.747,5.725,148.336
C02764=1232.998,161.341,-52.354,-177.749,5.724,148.336
C02765=1233.003,161.092,-52.332,-177.751,5.723,148.337
C02766=1233.008,160.843,-52.310,-177.754,5.722,148.337
C02767=1233.013,160.593,-52.289,-177.756,5.721,148.338
C02768=1233.018,160.345,-52.267,-177.759,5.719,148.338
C02769=1233.023,160.076,-52.243,-177.762,5.718,148.339
C02770=1233.028,159.807,-52.221,-177.765,5.717,148.339
C02771=1233.033,159.537,-52.197,-177.767,5.715,148.340
C02772=1233.037,159.268,-52.173,-177.770,5.714,148.340
C02773=1233.042,159.020,-52.152,-177.772,5.713,148.341
C02774=1233.047,158.770,-52.131,-177.775,5.712,148.341
C02775=1233.051,158.521,-52.109,-177.778,5.710,148.342
C02776=1233.056,158.272,-52.087,-177.780,5.709,148.342
C02777=1233.061,158.024,-52.065,-177.783,5.708,148.343
C02778=1233.065,157.774,-52.044,-177.785,5.707,148.343
C02779=1233.070,157.525,-52.022,-177.788,5.705,148.344
C02780=1233.075,157.277,-52.001,-177.790,5.704,148.344
C02781=1233.079,157.027,-51.979,-177.793,5.702,148.344
C02782=1233.085,156.778,-51.958,-177.795,5.702,148.345
C02783=1233.090,156.529,-51.936,-177.798,5.701,148.345
C02784=1233.094,156.280,-51.914,-177.801,5.699,148.346
C02785=1233.099,156.031,-51.892,-177.803,5.698,148.346
C02786=1233.104,155.782,-51.871,-177.806,5.697,148.347
C02787=1233.107,155.533,-51.850,-177.808,5.696,148.347
C02788=1233.112,155.284,-51.828,-177.811,5.694,148.348
C02789=1233.117,155.035,-51.807,-177.813,5.693,148.348
C02790=1233.122,154.786,-51.785,-177.815,5.692,148.349
C02791=1233.127,154.537,-51.764,-177.819,5.691,148.349
C02792=1233.132,154.288,-51.742,-177.821,5.690,148.350
C02793=1233.136,154.039,-51.720,-177.824,5.688,148.350
C02794=1233.140,153.790,-51.700,-177.826,5.687,148.351
C02795=1233.145,153.541,-51.678,-177.829,5.685,148.351
C02796=1233.150,153.292,-51.657,-177.831,5.685,148.352
C02797=1233.155,153.042,-51.635,-177.833,5.684,148.352
C02798=1233.160,152.794,-51.614,-177.836,5.682,148.353
C02799=1233.165,152.544,-51.593,-177.839,5.681,148.353
C02800=1233.168,152.295,-51.571,-177.842,5.680,148.354
C02801=1233.173,152.046,-51.550,-177.844,5.679,148.354
C02802=1233.178,151.798,-51.529,-177.846,5.678,148.354
C02803=1233.184,151.548,-51.508,-177.849,5.676,148.355
C02804=1233.188,151.299,-51.486,-177.851,5.675,148.355
C02805=1233.192,151.050,-51.465,-177.854,5.674,148.356
C02806=1233.197,150.801,-51.444,-177.856,5.673,148.356
C02807=1233.202,150.552,-51.423,-177.859,5.672,148.357
C02808=1233.207,150.303,-51.401,-177.862,5.670,148.357
C02809=1233.211,150.054,-51.380,-177.864,5.670,148.358
C02810=1233.216,149.805,-51.358,-177.867,5.668,148.358
C02811=1233.221,149.556,-51.337,-177.870,5.667,148.359
C02812=1233.225,149.308,-51.316,-177.872,5.666,148.359
C02813=1233.230,149.058,-51.295,-177.874,5.664,148.360
C02814=1233.235,148.808,-51.274,-177.877,5.664,148.360
C02815=1233.240,148.560,-51.252,-177.880,5.662,148.361
C02816=1233.244,148.311,-51.232,-177.882,5.661,148.361
C02817=1233.249,148.062,-51.210,-177.884,5.660,148.362
C02818=1233.254,147.812,-51.189,-177.887,5.659,148.362
C02819=1233.258,147.563,-51.169,-177.890,5.658,148.363
C02820=1233.263,147.315,-51.147,-177.893,5.656,148.363
C02821=1233.268,147.065,-51.126,-177.895,5.655,148.364
C02822=1233.273,146.816,-51.106,-177.897,5.655,148.364
C02823=1233.277,146.568,-51.084,-177.900,5.653,148.365
C02824=1233.282,146.318,-51.063,-177.903,5.652,148.365
C02825=1233.286,146.069,-51.042,-177.905,5.651,148.366
C02826=1233.291,145.820,-51.021,-177.908,5.650,148.366
C02827=1233.296,145.571,-51.000,-177.910,5.649,148.367
C02828=1233.301,145.322,-50.979,-177.913,5.647,148.367
C02829=1233.306,145.073,-50.958,-177.915,5.646,148.368
C02830=1233.310,144.824,-50.937,-177.917,5.645,148.368
C02831=1233.315,144.574,-50.916,-177.921,5.644,148.369
C02832=1233.319,144.325,-50.895,-177.923,5.643,148.369
C02833=1233.324,144.077,-50.874,-177.925,5.642,148.370
C02834=1233.329,143.828,-50.853,-177.928,5.640,148.370
C02835=1233.334,143.579,-50.832,-177.930,5.639,148.371
C02836=1233.339,143.329,-50.811,-177.933,5.638,148.371
C02837=1233.343,143.080,-50.791,-177.936,5.637,148.372
C02838=1233.348,142.831,-50.769,-177.938,5.636,148.372
C02839=1233.352,142.582,-50.749,-177.941,5.635,148.373
C02840=1233.357,142.333,-50.728,-177.943,5.634,148.373
C02841=1233.362,142.084,-50.707,-177.946,5.633,148.374
C02842=1233.367,141.835,-50.686,-177.948,5.631,148.374
C02843=1233.372,141.585,-50.665,-177.951,5.630,148.375
C02844=1233.376,141.337,-50.644,-177.953,5.629,148.375
C02845=1233.381,141.088,-50.623,-177.956,5.628,148.376
C02846=1233.386,140.839,-50.603,-177.958,5.627,148.376
C02847=1233.391,140.590,-50.582,-177.961,5.626,148.377
C02848=1233.395,140.340,-50.561,-177.964,5.624,148.377
C02849=1233.400,140.091,-50.540,-177.966,5.624,148.378
C02850=1233.404,139.842,-50.520,-177.968,5.623,148.378
C02851=1233.409,139.593,-50.500,-177.971,5.621,148.379
C02852=1233.414,139.344,-50.479,-177.974,5.620,148.379
C02853=1233.418,139.095,-50.458,-177.976,5.620,148.380
C02854=1233.424,138.845,-50.437,-177.979,5.618,148.380
C02855=1233.428,138.596,-50.417,-177.981,5.617,148.381
C02856=1233.433,138.347,-50.396,-177.984,5.616,148.381
C02857=1233.438,138.098,-50.376,-177.987,5.615,148.382
C02858=1233.443,137.849,-50.355,-177.989,5.614,148.382
C02859=1233.447,137.600,-50.334,-177.991,5.613,148.383
C02860=1233.452,137.351,-50.314,-177.995,5.612,148.384
C02861=1233.457,137.102,-50.293,-177.997,5.611,148.384
C02862=1233.461,136.853,-50.273,-177.999,5.610,148.385
C02863=1233.466,136.604,-50.252,-178.002,5.608,148.385
C02864=1233.471,136.355,-50.231,-178.005,5.608,148.386
C02865=1233.475,136.106,-50.211,-178.007,5.607,148.386
C02866=1233.481,135.856,-50.190,-178.010,5.605,148.387
C02867=1233.485,135.607,-50.169,-178.012,5.604,148.387
C02868=1233.489,135.359,-50.149,-178.015,5.603,148.388
C02869=1233.495,135.109,-50.128,-178.017,5.602,148.388
C02870=1233.499,134.860,-50.108,-178.020,5.601,148.389
C02871=1233.505,134.610,-50.088,-178.022,5.600,148.389
C02872=1233.509,134.361,-50.067,-178.025,5.599,148.390
C02873=1233.514,134.093,-50.045,-178.028,5.598,148.390
C02874=1233.518,133.824,-50.023,-178.030,5.597,148.391
C02875=1233.524,133.555,-50.001,-178.033,5.595,148.391
C02876=1233.529,133.287,-49.978,-178.036,5.595,148.392
C02877=1233.534,133.038,-49.958,-178.038,5.593,148.392
C02878=1233.538,132.789,-49.938,-178.041,5.592,148.393
C02879=1233.544,132.539,-49.918,-178.043,5.592,148.394
C02880=1233.548,132.290,-49.897,-178.046,5.590,148.394
C02881=1233.553,132.041,-49.877,-178.049,5.589,148.395
C02882=1233.558,131.792,-49.857,-178.051,5.588,148.395
C02883=1233.562,131.543,-49.836,-178.054,5.587,148.396
C02884=1233.567,131.294,-49.816,-178.056,5.586,148.396
C02885=1233.572,131.045,-49.796,-178.059,5.585,148.397
C02886=1233.577,130.796,-49.776,-178.061,5.584,148.397
C02887=1233.582,130.547,-49.755,-178.064,5.583,148.398
C02888=1233.586,130.298,-49.735,-178.067,5.582,148.398
C02889=1233.591,130.049,-49.714,-178.069,5.581,148.399
C02890=1233.595,129.799,-49.695,-178.072,5.580,148.399
C02891=1233.601,129.550,-49.674,-178.074,5.579,148.400
C02892=1233.605,129.301,-49.653,-178.077,5.578,148.400
C02893=1233.610,129.051,-49.634,-178.079,5.577,148.401
C02894=1233.614,128.802,-49.613,-178.082,5.576,148.402
C02895=1233.619,128.554,-49.593,-178.084,5.575,148.402
C02896=1233.625,128.304,-49.573,-178.087,5.574,148.403
C02897=1233.629,128.055,-49.553,-178.089,5.573,148.403
C02898=1233.634,127.806,-49.532,-178.092,5.571,148.404
C02899=1233.638,127.557,-49.513,-178.094,5.571,148.404
C02900=1233.643,127.308,-49.492,-178.097,5.570,148.405
C02901=1233.648,127.058,-49.473,-178.100,5.568,148.405
C02902=1233.653,126.809,-49.452,-178.102,5.568,148.406
C02903=1233.658,126.561,-49.432,-178.104,5.567,148.406
C02904=1233.663,126.311,-49.412,-178.107,5.566,148.407
C02905=1233.667,126.062,-49.392,-178.110,5.564,148.407
C02906=1233.672,125.813,-49.372,-178.112,5.564,148.408
C02907=1233.676,125.564,-49.352,-178.114,5.563,148.408
C02908=1233.681,125.314,-49.332,-178.117,5.562,148.409
C02909=1233.686,125.066,-49.312,-178.120,5.561,148.410
C02910=1233.691,124.816,-49.292,-178.122,5.560,148.410
C02911=1233.696,124.567,-49.271,-178.125,5.559,148.411
C02912=1233.701,124.317,-49.252,-178.127,5.558,148.411
C02913=1233.705,124.069,-49.231,-178.130,5.557,148.412
C02914=1233.710,123.820,-49.212,-178.133,5.556,148.412
C02915=1233.715,123.571,-49.192,-178.135,5.555,148.413
C02916=1233.720,123.321,-49.172,-178.138,5.554,148.413
C02917=1233.724,123.072,-49.152,-178.140,5.552,148.414
C02918=1233.729,122.823,-49.132,-178.143,5.552,148.414
C02919=1233.734,122.574,-49.112,-178.145,5.551,148.415
C02920=1233.739,122.325,-49.092,-178.148,5.550,148.415
C02921=1233.743,122.075,-49.073,-178.151,5.549,148.416
C02922=1233.748,121.826,-49.052,-178.153,5.548,148.416
C02923=1233.752,121.577,-49.033,-178.155,5.547,148.417
C02924=1233.757,121.329,-49.013,-178.158,5.546,148.418
C02925=1233.762,121.079,-48.993,-178.160,5.546,148.418
C02926=1233.767,120.829,-48.973,-178.163,5.544,148.419
C02927=1233.771,120.580,-48.953,-178.165,5.543,148.419
C02928=1233.777,120.332,-48.934,-178.168,5.542,148.420
C02929=1233.781,120.082,-48.914,-178.171,5.542,148.420
C02930=1233.786,119.833,-48.894,-178.173,5.540,148.421
C02931=1233.791,119.583,-48.874,-178.176,5.539,148.421
C02932=1233.796,119.335,-48.855,-178.179,5.539,148.422
C02933=1233.800,119.086,-48.834,-178.181,5.538,148.423
C02934=1233.805,118.836,-48.815,-178.184,5.536,148.423
C02935=1233.811,118.587,-48.795,-178.186,5.535,148.424
C02936=1233.815,118.338,-48.775,-178.189,5.535,148.424
C02937=1233.820,118.089,-48.755,-178.191,5.534,148.425
C02938=1233.824,117.839,-48.736,-178.193,5.533,148.425
C02939=1233.829,117.591,-48.717,-178.196,5.532,148.426
C02940=1233.833,117.342,-48.697,-178.199,5.531,148.426
C02941=1233.838,117.092,-48.677,-178.201,5.530,148.427
C02942=1233.844,116.843,-48.658,-178.204,5.529,148.428
C02943=1233.848,116.594,-48.638,-178.206,5.528,148.428
C02944=1233.853,116.344,-48.618,-178.209,5.527,148.429
C02945=1233.858,116.096,-48.598,-178.212,5.526,148.429
C02946=1233.863,115.846,-48.579,-178.214,5.525,148.430
C02947=1233.867,115.597,-48.560,-178.216,5.525,148.430
C02948=1233.872,115.348,-48.540,-178.219,5.524,148.431
C02949=1233.877,115.099,-48.521,-178.222,5.522,148.431
C02950=1233.882,114.849,-48.501,-178.224,5.522,148.432
C02951=1233.887,114.601,-48.481,-178.227,5.521,148.433
C02952=1233.891,114.351,-48.461,-178.229,5.520,148.433
C02953=1233.896,114.102,-48.442,-178.232,5.519,148.434
C02954=1233.901,113.853,-48.423,-178.234,5.518,148.434
C02955=1233.906,113.603,-48.403,-178.237,5.517,148.435
C02956=1233.910,113.354,-48.384,-178.240,5.516,148.435
C02957=1233.916,113.105,-48.364,-178.242,5.515,148.436
C02958=1233.920,112.855,-48.345,-178.244,5.515,148.436
C02959=1233.924,112.606,-48.326,-178.248,5.513,148.437
C02960=1233.930,112.357,-48.306,-178.250,5.512,148.437
C02961=1233.934,112.108,-48.286,-178.252,5.512,148.438
C02962=1233.940,111.860,-48.267,-178.255,5.511,148.439
C02963=1233.944,111.610,-48.248,-178.257,5.510,148.439
C02964=1233.948,111.361,-48.228,-178.260,5.509,148.440
C02965=1233.954,111.112,-48.209,-178.263,5.508,148.440
C02966=1233.958,110.862,-48.189,-178.265,5.507,148.441
C02967=1233.963,110.614,-48.170,-178.267,5.506,148.441
C02968=1233.968,110.364,-48.151,-178.270,5.506,148.442
C02969=1233.972,110.115,-48.131,-178.272,5.505,148.443
C02970=1233.978,109.866,-48.112,-178.275,5.503,148.443
C02971=1233.982,109.616,-48.093,-178.278,5.503,148.444
C02972=1233.987,109.367,-48.074,-178.280,5.502,148.444
C02973=1233.992,109.117,-48.054,-178.283,5.501,148.445
C02974=1233.997,108.869,-48.036,-178.285,5.501,148.445
C02975=1234.002,108.619,-48.016,-178.287,5.500,148.446
C02976=1234.006,108.370,-47.996,-178.291,5.498,148.447
C02977=1234.012,108.102,-47.976,-178.293,5.497,148.447
C02978=1234.017,107.833,-47.955,-178.296,5.497,148.448
C02979=1234.021,107.565,-47.935,-178.299,5.495,148.448
C02980=1234.027,107.296,-47.914,-178.302,5.495,148.449
C02981=1234.032,107.047,-47.895,-178.304,5.494,148.449
C02982=1234.037,106.798,-47.875,-178.306,5.493,148.450
C02983=1234.041,106.549,-47.857,-178.309,5.493,148.451
C02984=1234.046,106.300,-47.837,-178.311,5.492,148.451
C02985=1234.051,106.050,-47.817,-178.314,5.490,148.452
C02986=1234.056,105.801,-47.799,-178.317,5.490,148.452
C02987=1234.061,105.551,-47.780,-178.319,5.489,148.453
C02988=1234.065,105.303,-47.761,-178.322,5.488,148.454
C02989=1234.070,105.053,-47.741,-178.324,5.487,148.454
C02990=1234.075,104.804,-47.722,-178.326,5.486,148.455
C02991=1234.080,104.554,-47.704,-178.329,5.486,148.455
C02992=1234.085,104.306,-47.684,-178.332,5.484,148.456
C02993=1234.089,104.056,-47.665,-178.335,5.484,148.457
C02994=1234.094,103.807,-47.646,-178.337,5.483,148.457
C02995=1234.099,103.558,-47.628,-178.340,5.482,148.458
C02996=1234.104,103.309,-47.608,-178.342,5.481,148.458
C02997=1234.109,103.060,-47.589,-178.344,5.480,148.459
C02998=1234.113,102.811,-47.570,-178.347,5.480,148.459
C02999=1234.119,102.561,-47.551,-178.350,5.478,148.460
C03000=1234.123,102.312,-47.532,-178.352,5.477,148.460
C03001=1234.128,102.063,-47.513,-178.355,5.477,148.461
C03002=1234.133,101.813,-47.495,-178.357,5.476,148.462
C03003=1234.138,101.564,-47.475,-178.360,5.476,148.462
C03004=1234.142,101.315,-47.456,-178.362,5.475,148.463
C03005=1234.148,101.065,-47.438,-178.365,5.474,148.463
C03006=1234.152,100.816,-47.419,-178.367,5.473,148.464
C03007=1234.157,100.567,-47.399,-178.370,5.472,148.464
C03008=1234.162,100.318,-47.381,-178.373,5.471,148.465
C03009=1234.167,100.069,-47.362,-178.375,5.470,148.466
C03010=1234.171,99.819,-47.344,-178.378,5.470,148.466
C03011=1234.176,99.570,-47.324,-178.380,5.469,148.467
C03012=1234.181,99.321,-47.305,-178.383,5.468,148.467
C03013=1234.186,99.071,-47.287,-178.385,5.468,148.468
C03014=1234.190,98.823,-47.268,-178.387,5.467,148.468
C03015=1234.195,98.573,-47.250,-178.391,5.465,148.469
C03016=1234.200,98.324,-47.230,-178.393,5.464,148.470
C03017=1234.205,98.075,-47.212,-178.396,5.464,148.470
C03018=1234.210,97.825,-47.193,-178.398,5.463,148.471
C03019=1234.214,97.577,-47.174,-178.401,5.462,148.471
C03020=1234.220,97.327,-47.155,-178.403,5.462,148.472
C03021=1234.224,97.078,-47.136,-178.405,5.461,148.473
C03022=1234.229,96.829,-47.118,-178.408,5.460,148.473
C03023=1234.234,96.580,-47.099,-178.411,5.459,148.474
C03024=1234.239,96.330,-47.081,-178.413,5.459,148.474
C03025=1234.244,96.081,-47.061,-178.416,5.457,148.475
C03026=1234.248,95.831,-47.043,-178.419,5.456,148.476
C03027=1234.253,95.582,-47.025,-178.421,5.456,148.476
C03028=1234.259,95.333,-47.006,-178.424,5.455,148.477
C03029=1234.263,95.083,-46.987,-178.426,5.454,148.477
C03030=1234.267,94.835,-46.969,-178.428,5.454,148.478
C03031=1234.273,94.585,-46.950,-178.431,5.453,148.479
C03032=1234.277,94.336,-46.931,-178.434,5.452,148.479
C03033=1234.282,94.087,-46.913,-178.436,5.451,148.480
C03034=1234.288,93.837,-46.894,-178.438,5.451,148.480
C03035=1234.292,93.588,-46.875,-178.441,5.450,148.481
C03036=1234.297,93.339,-46.857,-178.444,5.449,148.482
C03037=1234.302,93.090,-46.838,-178.446,5.448,148.482
C03038=1234.306,92.840,-46.820,-178.449,5.447,148.483
C03039=1234.311,92.591,-46.802,-178.452,5.447,148.483
C03040=1234.316,92.342,-46.783,-178.454,5.446,148.484
C03041=1234.321,92.092,-46.764,-178.456,5.445,148.484
C03042=1234.326,91.843,-46.746,-178.459,5.444,148.485
C03043=1234.330,91.594,-46.727,-178.462,5.444,148.486
C03044=1234.336,91.345,-46.709,-178.464,5.443,148.486
C03045=1234.340,91.095,-46.691,-178.466,5.442,148.487
C03046=1234.345,90.846,-46.672,-178.469,5.442,148.487
C03047=1234.350,90.597,-46.654,-178.472,5.441,148.488
C03048=1234.355,90.347,-46.635,-178.474,5.440,148.489
C03049=1234.360,90.098,-46.617,-178.477,5.439,148.489
C03050=1234.364,89.849,-46.598,-178.480,5.438,148.490
C03051=1234.369,89.600,-46.580,-178.482,5.437,148.490
C03052=1234.374,89.350,-46.562,-178.485,5.437,148.491
C03053=1234.379,89.101,-46.543,-178.487,5.436,148.491
C03054=1234.384,88.852,-46.525,-178.490,5.435,148.492
C03055=1234.389,88.603,-46.507,-178.492,5.435,148.493
C03056=1234.393,88.353,-46.488,-178.495,5.434,148.493
C03057=1234.398,88.104,-46.470,-178.497,5.433,148.494
C03058=1234.404,87.855,-46.452,-178.500,5.432,148.495
C03059=1234.408,87.606,-46.433,-178.502,5.432,148.495
C03060=1234.413,87.356,-46.415,-178.505,5.431,148.496
C03061=1234.417,87.107,-46.397,-178.507,5.431,148.497
C03062=1234.422,86.858,-46.379,-178.510,5.430,148.497
C03063=1234.427,86.609,-46.361,-178.512,5.429,148.498
C03064=1234.432,86.358,-46.342,-178.515,5.428,148.498
C03065=1234.437,86.110,-46.323,-178.517,5.428,148.499
C03066=1234.442,85.861,-46.305,-178.521,5.426,148.500
C03067=1234.447,85.612,-46.287,-178.523,5.425,148.500
C03068=1234.452,85.362,-46.269,-178.525,5.425,148.501
C03069=1234.456,85.112,-46.251,-178.528,5.424,148.501
C03070=1234.461,84.863,-46.233,-178.531,5.424,148.502
C03071=1234.466,84.614,-46.215,-178.533,5.423,148.502
C03072=1234.471,84.365,-46.196,-178.535,5.422,148.503
C03073=1234.476,84.115,-46.178,-178.538,5.421,148.504
C03074=1234.481,83.866,-46.160,-178.541,5.421,148.504
C03075=1234.486,83.616,-46.142,-178.543,5.420,148.505
C03076=1234.490,83.367,-46.124,-178.545,5.419,148.505
C03077=1234.495,83.118,-46.106,-178.548,5.419,148.506
C03078=1234.500,82.869,-46.088,-178.551,5.418,148.507
C03079=1234.505,82.620,-46.070,-178.553,5.418,148.507
C03080=1234.510,82.371,-46.052,-178.556,5.417,148.508
C03081=1234.515,82.102,-46.032,-178.558,5.416,148.509
C03082=1234.520,81.833,-46.013,-178.561,5.416,148.509
C03083=1234.526,81.565,-45.993,-178.564,5.414,148.510
C03084=1234.531,81.297,-45.974,-178.567,5.414,148.511
C03085=1234.536,81.047,-45.956,-178.569,5.413,148.511
C03086=1234.540,80.798,-45.938,-178.572,5.412,148.512
C03087=1234.545,80.549,-45.920,-178.574,5.412,148.512
C03088=1234.550,80.300,-45.902,-178.577,5.411,148.513
C03089=1234.555,80.051,-45.884,-178.580,5.410,148.514
C03090=1234.560,79.801,-45.866,-178.582,5.409,148.514
C03091=1234.565,79.552,-45.848,-178.584,5.409,148.515
C03092=1234.570,79.302,-45.830,-178.587,5.408,148.515
C03093=1234.575,79.053,-45.812,-178.590,5.408,148.516
C03094=1234.579,78.803,-45.794,-178.592,5.407,148.517
C03095=1234.584,78.554,-45.776,-178.594,5.406,148.517
C03096=1234.589,78.305,-45.758,-178.597,5.405,148.518
C03097=1234.593,78.056,-45.741,-178.600,5.405,148.518
C03098=1234.598,77.807,-45.723,-178.602,5.404,148.519
C03099=1234.604,77.557,-45.706,-178.605,5.404,148.520
C03100=1234.608,77.308,-45.688,-178.607,5.403,148.520
C03101=1234.613,77.059,-45.670,-178.610,5.402,148.521
C03102=1234.618,76.810,-45.652,-178.612,5.401,148.522
C03103=1234.623,76.561,-45.634,-178.615,5.401,148.522
C03104=1234.628,76.310,-45.616,-178.617,5.400,148.523
C03105=1234.633,76.061,-45.598,-178.620,5.400,148.524
C03106=1234.638,75.812,-45.580,-178.622,5.399,148.524
C03107=1234.643,75.563,-45.562,-178.625,5.398,148.525
C03108=1234.647,75.314,-45.545,-178.627,5.397,148.525
C03109=1234.652,75.064,-45.527,-178.630,5.397,148.526
C03110=1234.657,74.815,-45.509,-178.633,5.396,148.527
C03111=1234.662,74.566,-45.491,-178.635,5.396,148.527
C03112=1234.667,74.316,-45.473,-178.637,5.395,148.528
C03113=1234.672,74.067,-45.456,-178.640,5.394,148.528
C03114=1234.677,73.817,-45.438,-178.643,5.394,148.529
C03115=1234.681,73.569,-45.421,-178.645,5.393,148.530
C03116=1234.686,73.319,-45.404,-178.648,5.392,148.530
C03117=1234.691,73.070,-45.386,-178.651,5.392,148.531
C03118=1234.696,72.820,-45.368,-178.653,5.391,148.531
C03119=1234.701,72.571,-45.350,-178.655,5.390,148.532
C03120=1234.706,72.321,-45.332,-178.658,5.390,148.533
C03121=1234.710,72.073,-45.315,-178.661,5.389,148.533
C03122=1234.716,71.823,-45.298,-178.663,5.388,148.534
C03123=1234.720,71.574,-45.280,-178.666,5.388,148.535
C03124=1234.725,71.324,-45.262,-178.668,5.387,148.535
C03125=1234.731,71.075,-45.244,-178.671,5.386,148.536
C03126=1234.735,70.826,-45.227,-178.673,5.386,148.536
C03127=1234.740,70.576,-45.210,-178.676,5.385,148.537
C03128=1234.745,70.327,-45.192,-178.679,5.385,148.538
C03129=1234.750,70.078,-45.174,-178.681,5.384,148.538
C03130=1234.754,69.828,-45.157,-178.684,5.383,148.539
C03131=1234.759,69.579,-45.139,-178.686,5.382,148.540
C03132=1234.764,69.329,-45.122,-178.689,5.382,148.540
C03133=1234.769,69.080,-45.104,-178.691,5.382,148.541
C03134=1234.774,68.830,-45.087,-178.693,5.381,148.542
C03135=1234.779,68.581,-45.069,-178.696,5.381,148.542
C03136=1234.784,68.331,-45.052,-178.699,5.380,148.543
C03137=1234.789,68.083,-45.035,-178.701,5.379,148.543
C03138=1234.794,67.834,-45.018,-178.703,5.379,148.544
C03139=1234.799,67.584,-45.000,-178.706,5.378,148.545
C03140=1234.803,67.335,-44.983,-178.709,5.378,148.545
C03141=1234.808,67.086,-44.965,-178.711,5.377,148.546
C03142=1234.813,66.836,-44.948,-178.714,5.376,148.547
C03143=1234.818,66.587,-44.930,-178.716,5.376,148.547
C03144=1234.823,66.337,-44.913,-178.719,5.375,148.548
C03145=1234.828,66.088,-44.895,-178.721,5.374,148.548
C03146=1234.832,65.839,-44.879,-178.724,5.374,148.549
C03147=1234.837,65.589,-44.861,-178.726,5.373,148.550
C03148=1234.842,65.340,-44.843,-178.729,5.372,148.550
C03149=1234.847,65.091,-44.827,-178.732,5.372,148.551
C03150=1234.852,64.842,-44.809,-178.734,5.371,148.552
C03151=1234.858,64.592,-44.792,-178.737,5.371,148.552
C03152=1234.862,64.343,-44.774,-178.739,5.370,148.553
C03153=1234.867,64.093,-44.757,-178.742,5.369,148.553
C03154=1234.872,63.843,-44.740,-178.744,5.369,148.554
C03155=1234.876,63.595,-44.722,-178.746,5.369,148.555
C03156=1234.882,63.345,-44.705,-178.749,5.368,148.555
C03157=1234.887,63.096,-44.689,-178.752,5.368,148.556
C03158=1234.892,62.847,-44.671,-178.754,5.367,148.557
C03159=1234.896,62.597,-44.654,-178.757,5.366,148.557
C03160=1234.901,62.347,-44.637,-178.759,5.366,148.558
C03161=1234.906,62.098,-44.619,-178.762,5.365,148.559
C03162=1234.911,61.849,-44.602,-178.764,5.364,148.559
C03163=1234.916,61.599,-44.585,-178.767,5.364,148.560
C03164=1234.921,61.351,-44.568,-178.770,5.363,148.561
C03165=1234.926,61.101,-44.551,-178.772,5.363,148.561
C03166=1234.930,60.852,-44.534,-178.775,5.362,148.562
C03167=1234.936,60.602,-44.517,-178.778,5.361,148.563
C03168=1234.940,60.353,-44.500,-178.780,5.360,148.563
C03169=1234.945,60.103,-44.482,-178.782,5.360,148.564
C03170=1234.950,59.854,-44.466,-178.784,5.360,148.564
C03171=1234.955,59.605,-44.449,-178.787,5.360,148.565
C03172=1234.960,59.355,-44.431,-178.790,5.359,148.566
C03173=1234.965,59.106,-44.414,-178.792,5.358,148.566
C03174=1234.970,58.856,-44.397,-178.795,5.358,148.567
C03175=1234.975,58.607,-44.380,-178.798,5.357,148.568
C03176=1234.979,58.358,-44.364,-178.800,5.357,148.568
C03177=1234.984,58.109,-44.346,-178.802,5.356,148.569
C03178=1234.989,57.859,-44.329,-178.805,5.355,148.569
C03179=1234.994,57.609,-44.312,-178.808,5.354,148.570
C03180=1234.999,57.361,-44.296,-178.810,5.354,148.571
C03181=1235.004,57.111,-44.278,-178.813,5.353,148.571
C03182=1235.009,56.861,-44.262,-178.815,5.354,148.572
C03183=1235.014,56.612,-44.244,-178.818,5.353,148.573
C03184=1235.019,56.363,-44.227,-178.820,5.352,148.573
C03185=1235.024,56.094,-44.209,-178.823,5.352,148.574
C03186=1235.030,55.826,-44.192,-178.825,5.351,148.575
C03187=1235.035,55.557,-44.173,-178.828,5.351,148.575
C03188=1235.040,55.289,-44.155,-178.831,5.350,148.576
C03189=1235.046,55.039,-44.138,-178.833,5.349,148.577
C03190=1235.050,54.791,-44.121,-178.836,5.349,148.577
C03191=1235.054,54.541,-44.104,-178.839,5.348,148.578
C03192=1235.060,54.292,-44.087,-178.841,5.348,148.579
C03193=1235.065,54.043,-44.070,-178.844,5.347,148.579
C03194=1235.069,53.793,-44.054,-178.847,5.347,148.580
C03195=1235.074,53.543,-44.036,-178.849,5.346,148.581
C03196=1235.079,53.295,-44.020,-178.851,5.345,148.581
C03197=1235.085,53.045,-44.003,-178.854,5.344,148.582
C03198=1235.089,52.795,-43.986,-178.856,5.345,148.583
C03199=1235.094,52.546,-43.969,-178.859,5.344,148.583
C03200=1235.099,52.297,-43.953,-178.861,5.344,148.584
C03201=1235.104,52.047,-43.936,-178.864,5.343,148.585
C03202=1235.108,51.798,-43.919,-178.867,5.342,148.585
C03203=1235.114,51.549,-43.902,-178.869,5.342,148.586
C03204=1235.119,51.299,-43.886,-178.872,5.341,148.587
C03205=1235.123,51.050,-43.869,-178.875,5.341,148.587
C03206=1235.128,50.801,-43.853,-178.877,5.340,148.588
C03207=1235.134,50.550,-43.836,-178.879,5.340,148.589
C03208=1235.138,50.301,-43.819,-178.881,5.339,148.589
C03209=1235.143,50.052,-43.803,-178.884,5.339,148.590
C03210=1235.148,49.802,-43.786,-178.887,5.338,148.590
C03211=1235.153,49.553,-43.769,-178.889,5.338,148.591
C03212=1235.158,49.304,-43.753,-178.892,5.337,148.592
C03213=1235.163,49.055,-43.736,-178.895,5.337,148.592
C03214=1235.168,48.805,-43.719,-178.897,5.336,148.593
C03215=1235.173,48.556,-43.703,-178.899,5.336,148.594
C03216=1235.178,48.306,-43.687,-178.902,5.336,148.594
C03217=1235.182,48.056,-43.670,-178.905,5.335,148.595
C03218=1235.188,47.807,-43.653,-178.907,5.334,148.596
C03219=1235.192,47.558,-43.637,-178.910,5.334,148.596
C03220=1235.197,47.309,-43.620,-178.912,5.333,148.597
C03221=1235.202,47.060,-43.604,-178.915,5.332,148.597
C03222=1235.207,46.809,-43.587,-178.917,5.332,148.598
C03223=1235.213,46.560,-43.571,-178.919,5.332,148.599
C03224=1235.217,46.311,-43.554,-178.922,5.332,148.600
C03225=1235.222,46.061,-43.537,-178.925,5.331,148.600
C03226=1235.227,45.813,-43.521,-178.927,5.330,148.601
C03227=1235.232,45.562,-43.505,-178.930,5.330,148.602
C03228=1235.237,45.313,-43.488,-178.932,5.329,148.602
C03229=1235.242,45.064,-43.472,-178.935,5.329,148.603
C03230=1235.246,44.814,-43.455,-178.937,5.329,148.604
C03231=1235.252,44.565,-43.439,-178.940,5.328,148.604
C03232=1235.256,44.316,-43.423,-178.942,5.328,148.605
C03233=1235.262,44.066,-43.406,-178.945,5.327,148.606
C03234=1235.267,43.816,-43.390,-178.948,5.327,148.606
C03235=1235.272,43.568,-43.373,-178.950,5.326,148.607
C03236=1235.276,43.318,-43.357,-178.953,5.325,148.607
C03237=1235.281,43.069,-43.340,-178.955,5.325,148.608
C03238=1235.286,42.819,-43.325,-178.957,5.325,148.609
C03239=1235.291,42.570,-43.308,-178.960,5.324,148.609
C03240=1235.296,42.321,-43.291,-178.962,5.324,148.610
C03241=1235.301,42.071,-43.275,-178.965,5.323,148.611
C03242=1235.306,41.822,-43.259,-178.968,5.322,148.611
C03243=1235.311,41.572,-43.243,-178.970,5.323,148.612
C03244=1235.316,41.323,-43.226,-178.972,5.322,148.613
C03245=1235.321,41.073,-43.210,-178.975,5.322,148.613
C03246=1235.326,40.824,-43.194,-178.978,5.321,148.614
C03247=1235.330,40.575,-43.178,-178.980,5.320,148.615
C03248=1235.335,40.324,-43.162,-178.983,5.320,148.615
C03249=1235.340,40.076,-43.145,-178.986,5.319,148.616
C03250=1235.345,39.826,-43.129,-178.988,5.320,148.617
C03251=1235.350,39.577,-43.113,-178.990,5.319,148.617
C03252=1235.355,39.327,-43.096,-178.993,5.318,148.618
C03253=1235.361,39.078,-43.080,-178.996,5.318,148.619
C03254=1235.365,38.828,-43.063,-178.998,5.317,148.620
C03255=1235.371,38.579,-43.048,-179.001,5.317,148.620
C03256=1235.375,38.329,-43.031,-179.003,5.317,148.621
C03257=1235.380,38.080,-43.016,-179.005,5.316,148.621
C03258=1235.385,37.830,-42.999,-179.008,5.315,148.622
C03259=1235.390,37.581,-42.983,-179.010,5.315,148.623
C03260=1235.395,37.332,-42.967,-179.013,5.314,148.623
C03261=1235.400,37.082,-42.951,-179.016,5.314,148.624
C03262=1235.405,36.833,-42.935,-179.018,5.314,148.625
C03263=1235.410,36.583,-42.919,-179.020,5.313,148.625
C03264=1235.415,36.334,-42.903,-179.023,5.313,148.626
C03265=1235.420,36.084,-42.887,-179.026,5.312,148.627
C03266=1235.425,35.835,-42.870,-179.028,5.312,148.627
C03267=1235.430,35.585,-42.854,-179.030,5.312,148.628
C03268=1235.434,35.337,-42.839,-179.033,5.311,148.629
C03269=1235.439,35.087,-42.823,-179.036,5.311,148.629
C03270=1235.444,34.837,-42.807,-179.038,5.310,148.630
C03271=1235.449,34.588,-42.790,-179.041,5.310,148.631
C03272=1235.454,34.338,-42.775,-179.044,5.309,148.631
C03273=1235.459,34.090,-42.759,-179.046,5.309,148.632
C03274=1235.464,33.840,-42.743,-179.048,5.309,148.633
C03275=1235.469,33.590,-42.727,-179.051,5.308,148.633
C03276=1235.474,33.341,-42.710,-179.054,5.308,148.634
C03277=1235.479,33.091,-42.695,-179.056,5.307,148.635
C03278=1235.484,32.842,-42.678,-179.058,5.307,148.636
C03279=1235.489,32.592,-42.662,-179.061,5.307,148.636
C03280=1235.494,32.343,-42.647,-179.064,5.306,148.637
C03281=1235.498,32.094,-42.631,-179.066,5.306,148.638
C03282=1235.504,31.844,-42.615,-179.069,5.305,148.638
C03283=1235.509,31.594,-42.599,-179.071,5.305,148.639
C03284=1235.514,31.345,-42.584,-179.074,5.305,148.640
C03285=1235.519,31.096,-42.567,-179.076,5.304,148.640
C03286=1235.524,30.846,-42.551,-179.079,5.304,148.641
C03287=1235.529,30.597,-42.536,-179.082,5.303,148.642
C03288=1235.533,30.348,-42.520,-179.083,5.303,148.642
C03289=1235.538,30.079,-42.503,-179.086,5.303,148.643
C03290=1235.544,29.811,-42.486,-179.089,5.302,148.644
C03291=1235.550,29.542,-42.469,-179.092,5.302,148.644
C03292=1235.555,29.274,-42.452,-179.094,5.301,148.645
C03293=1235.560,29.023,-42.436,-179.097,5.301,148.646
C03294=1235.565,28.774,-42.421,-179.100,5.300,148.646
C03295=1235.570,28.525,-42.405,-179.102,5.300,148.647
C03296=1235.575,28.275,-42.389,-179.104,5.300,148.648
C03297=1235.580,28.026,-42.373,-179.107,5.299,148.648
C03298=1235.585,27.777,-42.357,-179.110,5.299,148.649
C03299=1235.589,27.527,-42.342,-179.112,5.298,148.650
C03300=1235.595,27.277,-42.326,-179.114,5.298,148.650
C03301=1235.600,27.028,-42.311,-179.117,5.298,148.651
C03302=1235.604,26.779,-42.294,-179.120,5.297,148.652
C03303=1235.610,26.529,-42.279,-179.122,5.297,148.652
C03304=1235.615,26.280,-42.264,-179.125,5.296,148.653
C03305=1235.619,26.030,-42.248,-179.127,5.296,148.654
C03306=1235.625,25.781,-42.232,-179.130,5.296,148.655
C03307=1235.629,25.531,-42.217,-179.132,5.295,148.655
C03308=1235.634,25.281,-42.201,-179.135,5.295,148.656
C03309=1235.640,25.032,-42.185,-179.137,5.294,148.657
C03310=1235.645,24.783,-42.169,-179.140,5.295,148.657
C03311=1235.649,24.534,-42.154,-179.142,5.294,148.658
C03312=1235.654,24.284,-42.138,-179.145,5.293,148.659
C03313=1235.659,24.035,-42.123,-179.147,5.293,148.659
C03314=1235.664,23.786,-42.108,-179.150,5.293,148.660
C03315=1235.669,23.535,-42.092,-179.152,5.293,148.661
C03316=1235.674,23.286,-42.076,-179.155,5.292,148.661
C03317=1235.680,23.037,-42.061,-179.158,5.291,148.662
C03318=1235.684,22.788,-42.046,-179.160,5.291,148.663
C03319=1235.689,22.537,-42.030,-179.162,5.291,148.663
C03320=1235.694,22.288,-42.014,-179.165,5.291,148.664
C03321=1235.699,22.039,-41.999,-179.168,5.290,148.665
C03322=1235.704,21.790,-41.983,-179.170,5.289,148.665
C03323=1235.709,21.540,-41.968,-179.172,5.290,148.666
C03324=1235.714,21.290,-41.952,-179.175,5.289,148.667
C03325=1235.719,21.041,-41.937,-179.178,5.289,148.667
C03326=1235.724,20.792,-41.922,-179.180,5.288,148.668
C03327=1235.729,20.542,-41.906,-179.182,5.288,148.669
C03328=1235.734,20.292,-41.890,-179.185,5.288,148.670
C03329=1235.739,20.043,-41.875,-179.188,5.287,148.670
C03330=1235.744,19.794,-41.860,-179.190,5.287,148.671
C03331=1235.748,19.544,-41.844,-179.192,5.287,148.672
C03332=1235.754,19.295,-41.829,-179.195,5.286,148.672
C03333=1235.759,19.045,-41.813,-179.198,5.286,148.673
C03334=1235.764,18.796,-41.799,-179.200,5.285,148.674
C03335=1235.769,18.546,-41.783,-179.202,5.286,148.674
C03336=1235.773,18.296,-41.768,-179.205,5.285,148.675
C03337=1235.779,18.047,-41.752,-179.208,5.284,148.676
C03338=1235.783,17.798,-41.737,-179.210,5.284,148.676
C03339=1235.789,17.548,-41.722,-179.212,5.284,148.677
C03340=1235.794,17.299,-41.706,-179.215,5.284,148.678
C03341=1235.798,17.049,-41.691,-179.218,5.283,148.678
C03342=1235.804,16.799,-41.676,-179.220,5.283,148.679
C03343=1235.809,16.550,-41.661,-179.222,5.283,148.680
C03344=1235.814,16.301,-41.645,-179.225,5.282,148.680
C03345=1235.819,16.052,-41.630,-179.228,5.282,148.681
C03346=1235.824,15.802,-41.615,-179.230,5.281,148.682
C03347=1235.828,15.552,-41.599,-179.232,5.281,148.683
C03348=1235.834,15.302,-41.585,-179.235,5.281,148.683
C03349=1235.838,15.053,-41.570,-179.238,5.280,148.684
C03350=1235.844,14.804,-41.554,-179.240,5.280,148.685
C03351=1235.848,14.555,-41.539,-179.242,5.280,148.685
C03352=1235.854,14.305,-41.524,-179.245,5.280,148.686
C03353=1235.858,14.055,-41.509,-179.248,5.279,148.687
C03354=1235.864,13.806,-41.493,-179.250,5.278,148.687
C03355=1235.868,13.557,-41.478,-179.252,5.279,148.688
C03356=1235.874,13.306,-41.463,-179.256,5.279,148.689
C03357=1235.879,13.057,-41.448,-179.258,5.278,148.690
C03358=1235.884,12.808,-41.433,-179.261,5.277,148.690
C03359=1235.889,12.559,-41.418,-179.263,5.278,148.691
C03360=1235.894,12.309,-41.404,-179.266,5.277,148.692
C03361=1235.898,12.059,-41.388,-179.268,5.277,148.692
C03362=1235.903,11.810,-41.373,-179.270,5.277,148.693
C03363=1235.909,11.560,-41.358,-179.273,5.276,148.694
C03364=1235.913,11.311,-41.343,-179.276,5.276,148.694
C03365=1235.919,11.061,-41.327,-179.278,5.275,148.695
C03366=1235.924,10.812,-41.313,-179.280,5.276,148.696
C03367=1235.928,10.563,-41.298,-179.283,5.275,148.696
C03368=1235.934,10.313,-41.282,-179.286,5.274,148.697
C03369=1235.939,10.064,-41.268,-179.288,5.274,148.698
C03370=1235.944,9.814,-41.252,-179.290,5.274,148.699
C03371=1235.949,9.564,-41.238,-179.293,5.274,148.699
C03372=1235.953,9.315,-41.223,-179.296,5.273,148.700
C03373=1235.958,9.065,-41.207,-179.298,5.273,148.701
C03374=1235.963,8.816,-41.193,-179.300,5.273,148.701
C03375=1235.968,8.566,-41.178,-179.303,5.272,148.702
C03376=1235.974,8.316,-41.163,-179.306,5.272,148.703
C03377=1235.978,8.067,-41.148,-179.308,5.272,148.703
C03378=1235.983,7.818,-41.133,-179.310,5.271,148.704
C03379=1235.989,7.568,-41.118,-179.313,5.271,148.705
C03380=1235.993,7.319,-41.103,-179.315,5.271,148.705
C03381=1235.998,7.069,-41.089,-179.318,5.271,148.706
C03382=1236.004,6.820,-41.073,-179.320,5.270,148.707
C03383=1236.009,6.570,-41.059,-179.323,5.270,148.707
C03384=1236.013,6.321,-41.044,-179.325,5.270,148.708
C03385=1236.019,6.071,-41.029,-179.328,5.269,148.709
C03386=1236.024,5.822,-41.014,-179.330,5.269,148.709
C03387=1236.029,5.572,-41.000,-179.333,5.269,148.710
C03388=1236.034,5.323,-40.984,-179.335,5.269,148.711
C03389=1236.039,5.073,-40.970,-179.338,5.268,148.712
C03390=1236.044,4.824,-40.955,-179.340,5.267,148.712
C03391=1236.049,4.574,-40.941,-179.343,5.268,148.713
C03392=1236.054,4.325,-40.925,-179.346,5.268,148.714
C03393=1236.059,4.056,-40.909,-179.348,5.267,148.715
C03394=1236.064,3.788,-40.894,-179.351,5.266,148.715
C03395=1236.070,3.518,-40.877,-179.353,5.267,148.716
C03396=1236.075,3.250,-40.862,-179.356,5.267,148.717
C03397=1236.080,3.000,-40.847,-179.359,5.266,148.718
C03398=1236.085,2.750,-40.833,-179.362,5.266,148.718
C03399=1236.090,2.501,-40.818,-179.364,5.266,148.719
C03400=1236.095,2.251,-40.803,-179.366,5.265,148.720
C03401=1236.100,2.002,-40.788,-179.369,5.265,148.720
C03402=1236.105,1.752,-40.774,-179.371,5.265,148.721
C03403=1236.111,1.502,-40.759,-179.374,5.264,148.722
C03404=1236.115,1.253,-40.744,-179.376,5.264,148.722
C03405=1236.120,1.003,-40.730,-179.379,5.263,148.723
C03406=1236.125,0.754,-40.716,-179.381,5.264,148.724
C03407=1236.130,0.505,-40.701,-179.384,5.263,148.724
C03408=1236.135,0.255,-40.686,-179.386,5.263,148.725
C03409=1236.141,0.005,-40.671,-179.388,5.263,148.726
C03410=1236.146,-0.243,-40.657,-179.391,5.262,148.726
C03411=1236.151,-0.493,-40.643,-179.394,5.262,148.727
C03412=1236.156,-0.743,-40.628,-179.396,5.262,148.728
C03413=1236.160,-0.992,-40.613,-179.398,5.262,148.729
C03414=1236.165,-1.242,-40.599,-179.401,5.261,148.729
C03415=1236.171,-1.492,-40.584,-179.403,5.261,148.730
C03416=1236.176,-1.741,-40.570,-179.406,5.261,148.731
C03417=1236.181,-1.991,-40.555,-179.409,5.261,148.732
C03418=1236.186,-2.240,-40.541,-179.412,5.260,148.732
C03419=1236.191,-2.490,-40.526,-179.414,5.260,148.733
C03420=1236.196,-2.740,-40.512,-179.416,5.260,148.734
C03421=1236.200,-2.989,-40.497,-179.419,5.259,148.734
C03422=1236.206,-3.238,-40.483,-179.421,5.260,148.735
C03423=1236.211,-3.487,-40.469,-179.424,5.259,148.736
C03424=1236.216,-3.737,-40.454,-179.426,5.259,148.736
C03425=1236.221,-3.987,-40.439,-179.428,5.259,148.737
C03426=1236.226,-4.236,-40.425,-179.431,5.258,148.738
C03427=1236.231,-4.486,-40.410,-179.434,5.258,148.738
C03428=1236.236,-4.736,-40.396,-179.436,5.258,148.739
C03429=1236.241,-4.985,-40.382,-179.439,5.257,148.740
C03430=1236.246,-5.234,-40.368,-179.441,5.257,148.741
C03431=1236.251,-5.484,-40.353,-179.443,5.257,148.741
C03432=1236.256,-5.733,-40.339,-179.446,5.257,148.742
C03433=1236.261,-5.983,-40.324,-179.449,5.256,148.743
C03434=1236.266,-6.233,-40.310,-179.451,5.256,148.743
C03435=1236.271,-6.482,-40.296,-179.454,5.256,148.744
C03436=1236.276,-6.732,-40.282,-179.456,5.256,148.745
C03437=1236.281,-6.981,-40.268,-179.459,5.256,148.746
C03438=1236.286,-7.231,-40.253,-179.461,5.256,148.746
C03439=1236.291,-7.480,-40.238,-179.464,5.255,148.747
C03440=1236.296,-7.730,-40.224,-179.466,5.255,148.748
C03441=1236.301,-7.979,-40.210,-179.469,5.255,148.748
C03442=1236.306,-8.229,-40.196,-179.471,5.254,148.749
C03443=1236.311,-8.478,-40.182,-179.473,5.255,148.750
C03444=1236.316,-8.728,-40.167,-179.476,5.254,148.750
C03445=1236.321,-8.977,-40.153,-179.479,5.253,148.751
C03446=1236.326,-9.227,-40.139,-179.481,5.254,148.752
C03447=1236.331,-9.477,-40.125,-179.483,5.253,148.752
C03448=1236.336,-9.727,-40.110,-179.486,5.253,148.753
C03449=1236.342,-9.976,-40.096,-179.488,5.253,148.754
C03450=1236.347,-10.225,-40.082,-179.491,5.252,148.755
C03451=1236.352,-10.475,-40.068,-179.493,5.252,148.755
C03452=1236.357,-10.725,-40.054,-179.496,5.252,148.756
C03453=1236.362,-10.974,-40.039,-179.499,5.252,148.757
C03454=1236.367,-11.223,-40.025,-179.501,5.252,148.758
C03455=1236.372,-11.473,-40.011,-179.503,5.252,148.758
C03456=1236.377,-11.723,-39.997,-179.506,5.251,148.759
C03457=1236.381,-11.972,-39.983,-179.508,5.252,148.760
C03458=1236.387,-12.221,-39.969,-179.511,5.251,148.760
C03459=1236.392,-12.471,-39.955,-179.513,5.251,148.761
C03460=1236.397,-12.721,-39.941,-179.516,5.251,148.762
C03461=1236.402,-12.970,-39.926,-179.518,5.250,148.762
C03462=1236.407,-13.219,-39.912,-179.521,5.250,148.763
C03463=1236.412,-13.469,-39.898,-179.523,5.250,148.764
C03464=1236.417,-13.719,-39.885,-179.526,5.250,148.765
C03465=1236.422,-13.969,-39.870,-179.528,5.249,148.765
C03466=1236.427,-14.218,-39.857,-179.530,5.249,148.766
C03467=1236.432,-14.468,-39.843,-179.533,5.249,148.767
C03468=1236.437,-14.717,-39.828,-179.536,5.248,148.767
C03469=1236.442,-14.967,-39.814,-179.538,5.249,148.768
C03470=1236.448,-15.216,-39.800,-179.541,5.248,148.769
C03471=1236.453,-15.466,-39.786,-179.544,5.248,148.770
C03472=1236.458,-15.716,-39.772,-179.546,5.248,148.770
C03473=1236.462,-15.965,-39.759,-179.548,5.248,148.771
C03474=1236.468,-16.214,-39.745,-179.550,5.248,148.772
C03475=1236.473,-16.464,-39.731,-179.553,5.247,148.772
C03476=1236.477,-16.714,-39.716,-179.556,5.247,148.773
C03477=1236.483,-16.963,-39.702,-179.558,5.247,148.774
C03478=1236.488,-17.213,-39.689,-179.560,5.247,148.774
C03479=1236.493,-17.463,-39.675,-179.563,5.246,148.775
C03480=1236.498,-17.712,-39.661,-179.565,5.246,148.776
C03481=1236.503,-17.961,-39.647,-179.568,5.246,148.777
C03482=1236.508,-18.212,-39.633,-179.570,5.245,148.777
C03483=1236.513,-18.460,-39.620,-179.573,5.246,148.778
C03484=1236.518,-18.710,-39.606,-179.576,5.246,148.779
C03485=1236.523,-18.960,-39.592,-179.578,5.246,148.780
C03486=1236.529,-19.209,-39.578,-179.580,5.245,148.780
C03487=1236.533,-19.459,-39.565,-179.583,5.245,148.781
C03488=1236.538,-19.709,-39.550,-179.585,5.245,148.782
C03489=1236.544,-19.958,-39.536,-179.588,5.245,148.782
C03490=1236.549,-20.208,-39.523,-179.590,5.244,148.783
C03491=1236.553,-20.457,-39.509,-179.593,5.244,148.784
C03492=1236.559,-20.706,-39.495,-179.595,5.244,148.784
C03493=1236.564,-20.957,-39.482,-179.597,5.244,148.785
C03494=1236.569,-21.206,-39.467,-179.600,5.244,148.786
C03495=1236.574,-21.455,-39.454,-179.603,5.243,148.787
C03496=1236.579,-21.705,-39.441,-179.605,5.243,148.787
C03497=1236.584,-21.975,-39.426,-179.608,5.243,148.788
C03498=1236.590,-22.244,-39.411,-179.611,5.243,148.789
C03499=1236.596,-22.513,-39.396,-179.613,5.242,148.790
C03500=1236.601,-22.782,-39.382,-179.616,5.243,148.790
C03501=1236.605,-23.032,-39.367,-179.618,5.242,148.791
C03502=1236.611,-23.281,-39.353,-179.621,5.242,148.792
C03503=1236.616,-23.531,-39.340,-179.623,5.242,148.793
C03504=1236.621,-23.780,-39.326,-179.626,5.242,148.793
C03505=1236.626,-24.030,-39.313,-179.628,5.242,148.794
C03506=1236.631,-24.279,-39.299,-179.631,5.241,148.795
C03507=1236.636,-24.528,-39.285,-179.633,5.241,148.795
C03508=1236.641,-24.779,-39.272,-179.635,5.241,148.796
C03509=1236.646,-25.028,-39.258,-179.638,5.241,148.797
C03510=1236.652,-25.278,-39.245,-179.640,5.241,148.797
C03511=1236.656,-25.528,-39.231,-179.643,5.241,148.798
C03512=1236.662,-25.777,-39.218,-179.645,5.240,148.799
C03513=1236.667,-26.027,-39.204,-179.648,5.241,148.800
C03514=1236.672,-26.276,-39.191,-179.651,5.240,148.800
C03515=1236.677,-26.526,-39.177,-179.653,5.240,148.801
C03516=1236.682,-26.776,-39.163,-179.655,5.240,148.802
C03517=1236.687,-27.025,-39.150,-179.658,5.239,148.803
C03518=1236.692,-27.275,-39.136,-179.660,5.240,148.803
C03519=1236.697,-27.524,-39.123,-179.663,5.239,148.804
C03520=1236.702,-27.774,-39.110,-179.665,5.239,148.805
C03521=1236.707,-28.023,-39.096,-179.668,5.239,148.805
C03522=1236.712,-28.273,-39.083,-179.670,5.239,148.806
C03523=1236.718,-28.522,-39.069,-179.672,5.239,148.807
C03524=1236.722,-28.772,-39.056,-179.675,5.238,148.807
C03525=1236.727,-29.022,-39.042,-179.678,5.238,148.808
C03526=1236.732,-29.271,-39.029,-179.680,5.238,148.809
C03527=1236.737,-29.521,-39.015,-179.683,5.238,148.810
C03528=1236.742,-29.770,-39.002,-179.685,5.238,148.810
C03529=1236.748,-30.020,-38.989,-179.688,5.238,148.811
C03530=1236.752,-30.269,-38.975,-179.690,5.237,148.812
C03531=1236.758,-30.519,-38.962,-179.692,5.238,148.813
C03532=1236.763,-30.768,-38.948,-179.695,5.237,148.813
C03533=1236.768,-31.018,-38.935,-179.697,5.237,148.814
C03534=1236.773,-31.268,-38.922,-179.700,5.237,148.815
C03535=1236.778,-31.518,-38.908,-179.702,5.236,148.815
C03536=1236.783,-31.767,-38.895,-179.704,5.237,148.816
C03537=1236.788,-32.017,-38.881,-179.707,5.236,148.817
C03538=1236.793,-32.266,-38.868,-179.709,5.236,148.817
C03539=1236.798,-32.516,-38.855,-179.712,5.236,148.818
C03540=1236.803,-32.765,-38.842,-179.714,5.237,148.819
C03541=1236.808,-33.015,-38.828,-179.717,5.236,148.820
C03542=1236.814,-33.265,-38.815,-179.720,5.236,148.820
C03543=1236.818,-33.514,-38.801,-179.722,5.236,148.821
C03544=1236.824,-33.764,-38.788,-179.725,5.235,148.822
C03545=1236.829,-34.013,-38.775,-179.727,5.236,148.823
C03546=1236.834,-34.263,-38.762,-179.729,5.235,148.823
C03547=1236.840,-34.512,-38.748,-179.732,5.235,148.824
C03548=1236.844,-34.762,-38.735,-179.734,5.235,148.825
C03549=1236.849,-35.012,-38.723,-179.737,5.235,148.825
C03550=1236.854,-35.261,-38.709,-179.739,5.235,148.826
C03551=1236.859,-35.511,-38.696,-179.741,5.234,148.827
C03552=1236.865,-35.761,-38.682,-179.744,5.234,148.827
C03553=1236.870,-36.010,-38.670,-179.747,5.234,148.828
C03554=1236.874,-36.260,-38.656,-179.749,5.234,148.829
C03555=1236.880,-36.509,-38.643,-179.751,5.234,148.830
C03556=1236.885,-36.759,-38.630,-179.754,5.234,148.830
C03557=1236.890,-37.009,-38.617,-179.756,5.234,148.831
C03558=1236.895,-37.258,-38.604,-179.759,5.234,148.832
C03559=1236.899,-37.508,-38.590,-179.761,5.233,148.833
C03560=1236.905,-37.757,-38.577,-179.764,5.233,148.833
C03561=1236.910,-38.007,-38.565,-179.766,5.233,148.834
C03562=1236.916,-38.257,-38.551,-179.768,5.233,148.835
C03563=1236.921,-38.506,-38.539,-179.771,5.233,148.835
C03564=1236.925,-38.756,-38.526,-179.773,5.233,148.836
C03565=1236.931,-39.005,-38.512,-179.776,5.233,148.837
C03566=1236.936,-39.255,-38.499,-179.779,5.232,148.838
C03567=1236.941,-39.505,-38.486,-179.781,5.233,148.838
C03568=1236.946,-39.754,-38.473,-179.784,5.232,148.839
C03569=1236.951,-40.004,-38.460,-179.786,5.233,148.840
C03570=1236.956,-40.254,-38.447,-179.788,5.232,148.840
C03571=1236.962,-40.503,-38.434,-179.791,5.232,148.841
C03572=1236.966,-40.753,-38.420,-179.793,5.232,148.842
C03573=1236.971,-41.002,-38.408,-179.796,5.231,148.843
C03574=1236.976,-41.251,-38.395,-179.798,5.232,148.843
C03575=1236.982,-41.502,-38.382,-179.801,5.231,148.844
C03576=1236.987,-41.751,-38.369,-179.803,5.231,148.845
C03577=1236.991,-42.001,-38.356,-179.805,5.231,148.845
C03578=1236.997,-42.250,-38.343,-179.808,5.230,148.846
C03579=1237.002,-42.500,-38.330,-179.811,5.231,148.847
C03580=1237.007,-42.750,-38.317,-179.813,5.231,148.848
C03581=1237.012,-42.999,-38.305,-179.815,5.231,148.848
C03582=1237.018,-43.249,-38.292,-179.818,5.230,148.849
C03583=1237.022,-43.499,-38.279,-179.820,5.231,148.850
C03584=1237.027,-43.748,-38.266,-179.823,5.230,148.851
C03585=1237.033,-43.997,-38.253,-179.825,5.231,148.851
C03586=1237.038,-44.248,-38.240,-179.827,5.230,148.852
C03587=1237.043,-44.497,-38.227,-179.830,5.230,148.853
C03588=1237.048,-44.746,-38.215,-179.832,5.230,148.853
C03589=1237.053,-44.996,-38.202,-179.835,5.229,148.854
C03590=1237.058,-45.246,-38.189,-179.837,5.230,148.855
C03591=1237.064,-45.495,-38.176,-179.840,5.229,148.855
C03592=1237.069,-45.745,-38.163,-179.842,5.230,148.856
C03593=1237.073,-45.995,-38.150,-179.845,5.229,148.857
C03594=1237.078,-46.244,-38.138,-179.848,5.229,148.858
C03595=1237.083,-46.493,-38.125,-179.850,5.229,148.858
C03596=1237.089,-46.744,-38.112,-179.852,5.229,148.859
C03597=1237.094,-46.993,-38.099,-179.854,5.229,148.860
C03598=1237.099,-47.242,-38.086,-179.857,5.229,148.861
C03599=1237.104,-47.492,-38.074,-179.859,5.229,148.861
C03600=1237.109,-47.742,-38.061,-179.862,5.228,148.862
C03601=1237.115,-48.012,-38.048,-179.864,5.228,148.863
C03602=1237.120,-48.281,-38.034,-179.867,5.229,148.864
C03603=1237.125,-48.551,-38.020,-179.870,5.228,148.864
C03604=1237.132,-48.820,-38.006,-179.872,5.228,148.865
C03605=1237.136,-49.070,-37.993,-179.875,5.228,148.866
C03606=1237.141,-49.320,-37.981,-179.878,5.228,148.867
C03607=1237.146,-49.569,-37.968,-179.880,5.228,148.867
C03608=1237.151,-49.818,-37.956,-179.882,5.228,148.868
C03609=1237.156,-50.069,-37.943,-179.884,5.228,148.869
C03610=1237.162,-50.319,-37.930,-179.887,5.227,148.870
C03611=1237.167,-50.568,-37.917,-179.889,5.228,148.870
C03612=1237.172,-50.817,-37.905,-179.892,5.227,148.871
C03613=1237.177,-51.067,-37.892,-179.894,5.228,148.872
C03614=1237.182,-51.317,-37.880,-179.897,5.227,148.872
C03615=1237.188,-51.567,-37.867,-179.899,5.227,148.873
C03616=1237.193,-51.816,-37.855,-179.901,5.227,148.874
C03617=1237.197,-52.066,-37.842,-179.904,5.226,148.874
C03618=1237.202,-52.315,-37.829,-179.906,5.227,148.875
C03619=1237.208,-52.565,-37.817,-179.909,5.227,148.876
C03620=1237.213,-52.814,-37.805,-179.911,5.227,148.877
C03621=1237.218,-53.064,-37.792,-179.914,5.226,148.877
C03622=1237.222,-53.314,-37.779,-179.916,5.227,148.878
C03623=1237.228,-53.564,-37.767,-179.919,5.226,148.879
C03624=1237.234,-53.813,-37.754,-179.921,5.227,148.880
C03625=1237.239,-54.063,-37.742,-179.924,5.226,148.880
C03626=1237.244,-54.313,-37.730,-179.926,5.226,148.881
C03627=1237.249,-54.563,-37.717,-179.928,5.226,148.882
C03628=1237.254,-54.812,-37.704,-179.931,5.225,148.882
C03629=1237.259,-55.061,-37.691,-179.933,5.226,148.883
C03630=1237.265,-55.311,-37.680,-179.936,5.225,148.884
C03631=1237.270,-55.560,-37.667,-179.938,5.226,148.885
C03632=1237.274,-55.811,-37.654,-179.940,5.225,148.885
C03633=1237.280,-56.060,-37.642,-179.943,5.226,148.886
C03634=1237.285,-56.310,-37.630,-179.946,5.225,148.887
C03635=1237.289,-56.559,-37.618,-179.948,5.226,148.888
C03636=1237.295,-56.809,-37.606,-179.951,5.225,148.888
C03637=1237.300,-57.058,-37.593,-179.953,5.226,148.889
C03638=1237.304,-57.309,-37.581,-179.955,5.225,148.890
C03639=1237.310,-57.558,-37.568,-179.958,5.225,148.890
C03640=1237.315,-57.807,-37.556,-179.960,5.225,148.891
C03641=1237.320,-58.057,-37.544,-179.963,5.224,148.892
C03642=1237.325,-58.307,-37.531,-179.965,5.225,148.892
C03643=1237.330,-58.556,-37.518,-179.967,5.224,148.893
C03644=1237.336,-58.806,-37.507,-179.970,5.225,148.894
